LIN {X 0,Y 580.037,Z 775.595,A -85,B 0,C 180,E1 -1977.917,E2 -1977.917} C_VEL
LIN {X 0,Y 580.044,Z 776.896,A -85,B 0,C 180,E1 -1978.611,E2 -1978.611} C_VEL
LIN {X 0,Y 580.037,Z 777.71,A -85,B 0,C 180,E1 -1979.306,E2 -1979.306} C_VEL
LIN {X 0,Y 580.035,Z 777.996,A -85,B 0,C 180,E1 -1980,E2 -1980} C_VEL
LIN {X 0,Y 580.038,Z 777.754,A -85,B 0,C 180,E1 -1980.694,E2 -1980.694} C_VEL
LIN {X 0,Y 580.047,Z 777.018,A -85,B 0,C 180,E1 -1981.389,E2 -1981.389} C_VEL
LIN {X 0,Y 580.04,Z 775.802,A -85,B 0,C 180,E1 -1982.083,E2 -1982.083} C_VEL
LIN {X 0,Y 580.073,Z 772.961,A -85,B 0,C 180,E1 -1983.125,E2 -1983.125} C_VEL
LIN {X 0,Y 580.105,Z 768.85,A -85,B 0,C 180,E1 -1984.169,E2 -1984.169} C_VEL
LIN {X 0,Y 580.091,Z 763.255,A -85,B 0,C 180,E1 -1985.213,E2 -1985.213} C_VEL
LIN {X 0,Y 580.207,Z 757.174,A -85,B 0,C 180,E1 -1986.084,E2 -1986.084} C_VEL
LIN {X 0,Y 580.224,Z 749.516,A -85,B 0,C 180,E1 -1986.957,E2 -1986.957} C_VEL
LIN {X 0,Y 580.284,Z 740.89,A -85,B 0,C 180,E1 -1987.744,E2 -1987.744} C_VEL
LIN {X 0,Y 580.383,Z 731,A -85,B 0,C 180,E1 -1988.443,E2 -1988.443} C_VEL
LIN {X 0,Y 580.42,Z 721.403,A -85,B 0,C 180,E1 -1988.969,E2 -1988.969} C_VEL
LIN {X 0,Y 580.469,Z 711.987,A -85,B 0,C 180,E1 -1989.363,E2 -1989.363} C_VEL
LIN {X 0,Y 580.511,Z 701.019,A -85,B 0,C 180,E1 -1989.692,E2 -1989.692} C_VEL
LIN {X 0,Y 580.608,Z 688.344,A -85,B 0,C 180,E1 -1989.911,E2 -1989.911} C_VEL
LIN {X 0,Y 580.624,Z 626.629,A -85,B 0,C 180,E1 -1990.67,E2 -1990.67} C_VEL
LIN {X 0,Y 579.916,Z 622.77,A -85,B 0,C 180,E1 -1990.759,E2 -1990.759} C_VEL
LIN {X 0,Y 578.276,Z 619.333,A -85,B 0,C 180,E1 -1990.91,E2 -1990.91} C_VEL
LIN {X 0,Y 575.656,Z 615.329,A -85,B 0,C 180,E1 -1991.191,E2 -1991.191} C_VEL
LIN {X 0,Y 573.643,Z 611.693,A -85,B 0,C 180,E1 -1991.558,E2 -1991.558} C_VEL
LIN {X 0,Y 573.314,Z 609.974,A -85,B 0,C 180,E1 -1991.77,E2 -1991.77} C_VEL
LIN {X 0,Y 573.481,Z 588.417,A -85,B 0,C 180,E1 -1994.607,E2 -1994.607} C_VEL
LIN {X 0,Y 573.675,Z 565.715,A -85,B 0,C 180,E1 -1997.632,E2 -1997.632} C_VEL
LIN {X 0,Y 573.922,Z 545.049,A -85,B 0,C 180,E1 -2000.426,E2 -2000.426} C_VEL
LIN {X 0,Y 574.25,Z 522.477,A -85,B 0,C 180,E1 -2003.532,E2 -2003.532} C_VEL
LIN {X 0,Y 574.202,Z 517.675,A -85,B 0,C 180,E1 -2004.207,E2 -2004.207} C_VEL
LIN {X 0,Y 573.309,Z 513.19,A -85,B 0,C 180,E1 -2004.924,E2 -2004.924} C_VEL
LIN {X 0,Y 573.256,Z 513.08,A -85,B 0,C 180,E1 -2008.029,E2 -2008.029} C_VEL
LIN {X 0,Y 573.249,Z 513.077,A -85,B 0,C 180,E1 -2010.176,E2 -2010.176} C_VEL
LIN {X 0,Y 573.256,Z 513.073,A -85,B 0,C 180,E1 -2012.645,E2 -2012.645} C_VEL
LIN {X 0,Y 573.257,Z 513.076,A -85,B 0,C 180,E1 -2015.185,E2 -2015.185} C_VEL
LIN {X 0,Y 573.237,Z 513.08,A -85,B 0,C 180,E1 -2017.808,E2 -2017.808} C_VEL
LIN {X 0,Y 573.248,Z 513.07,A -85,B 0,C 180,E1 -2020.525,E2 -2020.525} C_VEL
LIN {X 0,Y 573.239,Z 513.077,A -85,B 0,C 180,E1 -2023.359,E2 -2023.359} C_VEL
LIN {X 0,Y 573.249,Z 513.073,A -85,B 0,C 180,E1 -2026.331,E2 -2026.331} C_VEL
LIN {X 0,Y 573.238,Z 513.074,A -85,B 0,C 180,E1 -2028.543,E2 -2028.543} C_VEL
LIN {X 0,Y 573.246,Z 513.081,A -85,B 0,C 180,E1 -2031.298,E2 -2031.298} C_VEL
LIN {X 0,Y 573.217,Z 513.077,A -85,B 0,C 180,E1 -2034.018,E2 -2034.018} C_VEL
LIN {X 0,Y 573.243,Z 513.075,A -85,B 0,C 180,E1 -2036.516,E2 -2036.516} C_VEL
LIN {X 0,Y 573.235,Z 513.084,A -85,B 0,C 180,E1 -2039.117,E2 -2039.117} C_VEL
LIN {X 0,Y 573.256,Z 513.073,A -85,B 0,C 180,E1 -2041.971,E2 -2041.971} C_VEL
LIN {X 0,Y 573.253,Z 513.079,A -85,B 0,C 180,E1 -2044.589,E2 -2044.589} C_VEL
LIN {X 0,Y 573.238,Z 513.075,A -85,B 0,C 180,E1 -2047.662,E2 -2047.662} C_VEL
LIN {X 0,Y 573.317,Z 513.261,A -85,B 0,C 180,E1 -2050.276,E2 -2050.276} C_VEL
LIN {X 0,Y 573.558,Z 518.552,A -85,B 0,C 180,E1 -2051.237,E2 -2051.237} C_VEL
LIN {X 0,Y 573.387,Z 536.372,A -85,B 0,C 180,E1 -2054.356,E2 -2054.356} C_VEL
LIN {X 0,Y 573.308,Z 547.196,A -85,B 0,C 180,E1 -2056.192,E2 -2056.192} C_VEL
LIN {X 0,Y 573.776,Z 550.138,A -85,B 0,C 180,E1 -2056.277,E2 -2056.277} C_VEL
LIN {X 0,Y 574.078,Z 556.843,A -85,B 0,C 180,E1 -2056.369,E2 -2056.369} C_VEL
LIN {X 0,Y 573.884,Z 653.915,A -85,B 0,C 180,E1 -2057.602,E2 -2057.602} C_VEL
LIN {X 0,Y 573.815,Z 667.201,A -85,B 0,C 180,E1 -2057.915,E2 -2057.915} C_VEL
LIN {X 0,Y 573.718,Z 679.36,A -85,B 0,C 180,E1 -2058.339,E2 -2058.339} C_VEL
LIN {X 0,Y 573.588,Z 690.955,A -85,B 0,C 180,E1 -2058.881,E2 -2058.881} C_VEL
LIN {X 0,Y 573.447,Z 702.546,A -85,B 0,C 180,E1 -2059.585,E2 -2059.585} C_VEL
LIN {X 0,Y 573.332,Z 713.058,A -85,B 0,C 180,E1 -2060.385,E2 -2060.385} C_VEL
LIN {X 0,Y 573.242,Z 721.659,A -85,B 0,C 180,E1 -2061.184,E2 -2061.184} C_VEL
LIN {X 0,Y 573.162,Z 729.583,A -85,B 0,C 180,E1 -2062.07,E2 -2062.07} C_VEL
LIN {X 0,Y 573.092,Z 737.519,A -85,B 0,C 180,E1 -2063.162,E2 -2063.162} C_VEL
LIN {X 0,Y 573.071,Z 744.447,A -85,B 0,C 180,E1 -2064.369,E2 -2064.369} C_VEL
LIN {X 0,Y 573.028,Z 749.189,A -85,B 0,C 180,E1 -2065.427,E2 -2065.427} C_VEL
LIN {X 0,Y 573.022,Z 752.822,A -85,B 0,C 180,E1 -2066.484,E2 -2066.484} C_VEL
LIN {X 0,Y 572.959,Z 754.699,A -85,B 0,C 180,E1 -2067.187,E2 -2067.187} C_VEL
LIN {X 0,Y 572.939,Z 756.128,A -85,B 0,C 180,E1 -2067.89,E2 -2067.89} C_VEL
LIN {X 0,Y 572.941,Z 757.755,A -85,B 0,C 180,E1 -2069.297,E2 -2069.297} C_VEL
LIN {X 0,Y 572.939,Z 757.996,A -85,B 0,C 180,E1 -2069.999,E2 -2069.999} C_VEL
LIN {X 0,Y 572.94,Z 757.815,A -85,B 0,C 180,E1 -2070.702,E2 -2070.702} C_VEL
LIN {X 0,Y 572.939,Z 756.273,A -85,B 0,C 180,E1 -2072.108,E2 -2072.108} C_VEL
LIN {X 0,Y 572.96,Z 754.912,A -85,B 0,C 180,E1 -2072.812,E2 -2072.812} C_VEL
LIN {X 0,Y 573.015,Z 752.034,A -85,B 0,C 180,E1 -2073.867,E2 -2073.867} C_VEL
LIN {X 0,Y 572.963,Z 748.134,A -85,B 0,C 180,E1 -2074.925,E2 -2074.925} C_VEL
LIN {X 0,Y 573.075,Z 743.102,A -85,B 0,C 180,E1 -2075.983,E2 -2075.983} C_VEL
LIN {X 0,Y 573.082,Z 736.781,A -85,B 0,C 180,E1 -2077.044,E2 -2077.044} C_VEL
LIN {X 0,Y 573.177,Z 728.86,A -85,B 0,C 180,E1 -2078.105,E2 -2078.105} C_VEL
LIN {X 0,Y 573.286,Z 719.011,A -85,B 0,C 180,E1 -2079.17,E2 -2079.17} C_VEL
LIN {X 0,Y 573.424,Z 708.694,A -85,B 0,C 180,E1 -2080.058,E2 -2080.058} C_VEL
LIN {X 0,Y 573.556,Z 697.058,A -85,B 0,C 180,E1 -2080.858,E2 -2080.858} C_VEL
LIN {X 0,Y 573.657,Z 686.212,A -85,B 0,C 180,E1 -2081.449,E2 -2081.449} C_VEL
LIN {X 0,Y 573.754,Z 673.632,A -85,B 0,C 180,E1 -2081.969,E2 -2081.969} C_VEL
LIN {X 0,Y 573.845,Z 660.474,A -85,B 0,C 180,E1 -2082.353,E2 -2082.353} C_VEL
LIN {X 0,Y 573.912,Z 648.141,A -85,B 0,C 180,E1 -2082.576,E2 -2082.576} C_VEL
LIN {X 0,Y 573.917,Z 551.106,A -85,B 0,C 180,E1 -2083.798,E2 -2083.798} C_VEL
LIN {X 0,Y 573.364,Z 547.542,A -85,B 0,C 180,E1 -2083.873,E2 -2083.873} C_VEL
LIN {X 0,Y 573.298,Z 546.336,A -85,B 0,C 180,E1 -2084.011,E2 -2084.011} C_VEL
LIN {X 0,Y 573.451,Z 530.701,A -85,B 0,C 180,E1 -2086.721,E2 -2086.721} C_VEL
LIN {X 0,Y 573.578,Z 515.71,A -85,B 0,C 180,E1 -2089.356,E2 -2089.356} C_VEL
LIN {X 0,Y 573.272,Z 513.184,A -85,B 0,C 180,E1 -2089.841,E2 -2089.841} C_VEL
LIN {X 0,Y 573.238,Z 513.076,A -85,B 0,C 180,E1 -2092.337,E2 -2092.337} C_VEL
LIN {X 0,Y 573.256,Z 513.081,A -85,B 0,C 180,E1 -2095.409,E2 -2095.409} C_VEL
LIN {X 0,Y 573.253,Z 513.074,A -85,B 0,C 180,E1 -2098.028,E2 -2098.028} C_VEL
LIN {X 0,Y 573.239,Z 513.076,A -85,B 0,C 180,E1 -2100.883,E2 -2100.883} C_VEL
LIN {X 0,Y 573.261,Z 513.08,A -85,B 0,C 180,E1 -2103.523,E2 -2103.523} C_VEL
LIN {X 0,Y 573.259,Z 513.072,A -85,B 0,C 180,E1 -2106.047,E2 -2106.047} C_VEL
LIN {X 0,Y 573.247,Z 513.074,A -85,B 0,C 180,E1 -2108.7,E2 -2108.7} C_VEL
LIN {X 0,Y 573.252,Z 513.08,A -85,B 0,C 180,E1 -2111.595,E2 -2111.595} C_VEL
LIN {X 0,Y 573.236,Z 513.073,A -85,B 0,C 180,E1 -2114.332,E2 -2114.332} C_VEL
LIN {X 0,Y 573.236,Z 513.083,A -85,B 0,C 180,E1 -2117.358,E2 -2117.358} C_VEL
LIN {X 0,Y 573.246,Z 513.071,A -85,B 0,C 180,E1 -2120.393,E2 -2120.393} C_VEL
LIN {X 0,Y 573.251,Z 513.075,A -85,B 0,C 180,E1 -2123.077,E2 -2123.077} C_VEL
LIN {X 0,Y 573.27,Z 513.077,A -85,B 0,C 180,E1 -2125.671,E2 -2125.671} C_VEL
LIN {X 0,Y 573.245,Z 513.074,A -85,B 0,C 180,E1 -2128.185,E2 -2128.185} C_VEL
LIN {X 0,Y 573.265,Z 513.071,A -85,B 0,C 180,E1 -2130.634,E2 -2130.634} C_VEL
LIN {X 0,Y 573.265,Z 513.08,A -85,B 0,C 180,E1 -2133.5,E2 -2133.5} C_VEL
LIN {X 0,Y 573.227,Z 513.076,A -85,B 0,C 180,E1 -2136.134,E2 -2136.134} C_VEL
LIN {X 0,Y 573.256,Z 513.076,A -85,B 0,C 180,E1 -2139.174,E2 -2139.174} C_VEL
LIN {X 0,Y 573.233,Z 513.083,A -85,B 0,C 180,E1 -2141.411,E2 -2141.411} C_VEL
LIN {X 0,Y 573.253,Z 513.08,A -85,B 0,C 180,E1 -2143.622,E2 -2143.622} C_VEL
LIN {X 0,Y 573.229,Z 513.075,A -85,B 0,C 180,E1 -2146.529,E2 -2146.529} C_VEL
LIN {X 0,Y 573.255,Z 513.072,A -85,B 0,C 180,E1 -2148.745,E2 -2148.745} C_VEL
LIN {X 0,Y 573.301,Z 513.075,A -85,B 0,C 180,E1 -2151.541,E2 -2151.541} C_VEL
LIN {X 0,Y 573.285,Z 513.068,A -85,B 0,C 180,E1 -2154.372,E2 -2154.372} C_VEL
LIN {X 0,Y 573.303,Z 513.07,A -85,B 0,C 180,E1 -2157.892,E2 -2157.892} C_VEL
LIN {X 0,Y 573.33,Z 513.063,A -85,B 0,C 180,E1 -2160.702,E2 -2160.702} C_VEL
LIN {X 0,Y 573.234,Z 513.083,A -85,B 0,C 180,E1 -2163.514,E2 -2163.514} C_VEL
LIN {X 0,Y 573.284,Z 513.078,A -85,B 0,C 180,E1 -2165.628,E2 -2165.628} C_VEL
LIN {X 0,Y 573.285,Z 513.068,A -85,B 0,C 180,E1 -2168.459,E2 -2168.459} C_VEL
LIN {X 0,Y 573.264,Z 513.075,A -85,B 0,C 180,E1 -2171.312,E2 -2171.312} C_VEL
LIN {X 0,Y 573.266,Z 513.072,A -85,B 0,C 180,E1 -2174.193,E2 -2174.193} C_VEL
LIN {X 0,Y 573.252,Z 513.074,A -85,B 0,C 180,E1 -2177.112,E2 -2177.112} C_VEL
LIN {X 0,Y 573.249,Z 513.075,A -85,B 0,C 180,E1 -2180.077,E2 -2180.077} C_VEL
LIN {X 0,Y 573.231,Z 513.075,A -85,B 0,C 180,E1 -2182.338,E2 -2182.338} C_VEL
LIN {X 0,Y 573.251,Z 513.079,A -85,B 0,C 180,E1 -2185.41,E2 -2185.41} C_VEL
LIN {X 0,Y 573.258,Z 513.076,A -85,B 0,C 180,E1 -2188.032,E2 -2188.032} C_VEL
LIN {X 0,Y 573.232,Z 513.075,A -85,B 0,C 180,E1 -2190.885,E2 -2190.885} C_VEL
LIN {X 0,Y 573.283,Z 513.077,A -85,B 0,C 180,E1 -2193.529,E2 -2193.529} C_VEL
LIN {X 0,Y 573.256,Z 513.073,A -85,B 0,C 180,E1 -2196.049,E2 -2196.049} C_VEL
LIN {X 0,Y 573.244,Z 513.073,A -85,B 0,C 180,E1 -2198.702,E2 -2198.702} C_VEL
LIN {X 0,Y 573.249,Z 513.082,A -85,B 0,C 180,E1 -2201.596,E2 -2201.596} C_VEL
LIN {X 0,Y 573.231,Z 513.076,A -85,B 0,C 180,E1 -2204.334,E2 -2204.334} C_VEL
LIN {X 0,Y 573.248,Z 513.077,A -85,B 0,C 180,E1 -2207.358,E2 -2207.358} C_VEL
LIN {X 0,Y 573.245,Z 513.073,A -85,B 0,C 180,E1 -2210.394,E2 -2210.394} C_VEL
LIN {X 0,Y 573.254,Z 513.071,A -85,B 0,C 180,E1 -2213.079,E2 -2213.079} C_VEL
LIN {X 0,Y 573.266,Z 513.08,A -85,B 0,C 180,E1 -2215.672,E2 -2215.672} C_VEL
LIN {X 0,Y 573.248,Z 513.065,A -85,B 0,C 180,E1 -2218.186,E2 -2218.186} C_VEL
LIN {X 0,Y 573.263,Z 513.071,A -85,B 0,C 180,E1 -2220.635,E2 -2220.635} C_VEL
LIN {X 0,Y 573.251,Z 513.073,A -85,B 0,C 180,E1 -2223.025,E2 -2223.025} C_VEL
LIN {X 0,Y 573.275,Z 513.075,A -85,B 0,C 180,E1 -2225.367,E2 -2225.367} C_VEL
LIN {X 0,Y 573.287,Z 513.31,A -85,B 0,C 180,E1 -2226.936,E2 -2226.936} C_VEL
LIN {X 0,Y 574.008,Z 518.026,A -85,B 0,C 180,E1 -2227.695,E2 -2227.695} C_VEL
LIN {X 0,Y 573.748,Z 538.175,A -85,B 0,C 180,E1 -2230.688,E2 -2230.688} C_VEL
LIN {X 0,Y 573.546,Z 557.107,A -85,B 0,C 180,E1 -2233.454,E2 -2233.454} C_VEL
LIN {X 0,Y 573.395,Z 576.024,A -85,B 0,C 180,E1 -2236.15,E2 -2236.15} C_VEL
LIN {X 0,Y 574.056,Z 581.566,A -85,B 0,C 180,E1 -2236.257,E2 -2236.257} C_VEL
LIN {X 0,Y 573.882,Z 683.982,A -85,B 0,C 180,E1 -2237.558,E2 -2237.558} C_VEL
LIN {X 0,Y 573.811,Z 697.238,A -85,B 0,C 180,E1 -2237.871,E2 -2237.871} C_VEL
LIN {X 0,Y 573.718,Z 709.387,A -85,B 0,C 180,E1 -2238.295,E2 -2238.295} C_VEL
LIN {X 0,Y 573.576,Z 721.729,A -85,B 0,C 180,E1 -2238.879,E2 -2238.879} C_VEL
LIN {X 0,Y 573.438,Z 733.213,A -85,B 0,C 180,E1 -2239.586,E2 -2239.586} C_VEL
LIN {X 0,Y 573.327,Z 743.607,A -85,B 0,C 180,E1 -2240.386,E2 -2240.386} C_VEL
LIN {X 0,Y 573.24,Z 752.119,A -85,B 0,C 180,E1 -2241.185,E2 -2241.185} C_VEL
LIN {X 0,Y 573.16,Z 759.966,A -85,B 0,C 180,E1 -2242.072,E2 -2242.072} C_VEL
LIN {X 0,Y 573.072,Z 767.958,A -85,B 0,C 180,E1 -2243.186,E2 -2243.186} C_VEL
LIN {X 0,Y 573.07,Z 774.683,A -85,B 0,C 180,E1 -2244.37,E2 -2244.37} C_VEL
LIN {X 0,Y 573.028,Z 779.374,A -85,B 0,C 180,E1 -2245.428,E2 -2245.428} C_VEL
LIN {X 0,Y 573.022,Z 782.96,A -85,B 0,C 180,E1 -2246.485,E2 -2246.485} C_VEL
LIN {X 0,Y 572.959,Z 784.811,A -85,B 0,C 180,E1 -2247.188,E2 -2247.188} C_VEL
LIN {X 0,Y 572.937,Z 786.201,A -85,B 0,C 180,E1 -2247.892,E2 -2247.892} C_VEL
LIN {X 0,Y 572.94,Z 787.785,A -85,B 0,C 180,E1 -2249.298,E2 -2249.298} C_VEL
LIN {X 0,Y 572.938,Z 788,A -85,B 0,C 180,E1 -2250.001,E2 -2250.001} C_VEL
LIN {X 0,Y 572.946,Z 787.185,A -85,B 0,C 180,E1 -2251.406,E2 -2251.406} C_VEL
LIN {X 0,Y 572.937,Z 786.198,A -85,B 0,C 180,E1 -2252.11,E2 -2252.11} C_VEL
LIN {X 0,Y 572.959,Z 784.807,A -85,B 0,C 180,E1 -2252.813,E2 -2252.813} C_VEL
LIN {X 0,Y 573.014,Z 781.894,A -85,B 0,C 180,E1 -2253.869,E2 -2253.869} C_VEL
LIN {X 0,Y 572.963,Z 777.948,A -85,B 0,C 180,E1 -2254.926,E2 -2254.926} C_VEL
LIN {X 0,Y 573.064,Z 771.874,A -85,B 0,C 180,E1 -2256.161,E2 -2256.161} C_VEL
LIN {X 0,Y 573.12,Z 765.234,A -85,B 0,C 180,E1 -2257.221,E2 -2257.221} C_VEL
LIN {X 0,Y 573.201,Z 756.986,A -85,B 0,C 180,E1 -2258.284,E2 -2258.284} C_VEL
LIN {X 0,Y 573.287,Z 748.532,A -85,B 0,C 180,E1 -2259.171,E2 -2259.171} C_VEL
LIN {X 0,Y 573.409,Z 738.091,A -85,B 0,C 180,E1 -2260.059,E2 -2260.059} C_VEL
LIN {X 0,Y 573.55,Z 726.343,A -85,B 0,C 180,E1 -2260.858,E2 -2260.858} C_VEL
LIN {X 0,Y 573.654,Z 715.271,A -85,B 0,C 180,E1 -2261.448,E2 -2261.448} C_VEL
LIN {X 0,Y 573.767,Z 702.163,A -85,B 0,C 180,E1 -2261.974,E2 -2261.974} C_VEL
LIN {X 0,Y 573.836,Z 689.501,A -85,B 0,C 180,E1 -2262.332,E2 -2262.332} C_VEL
LIN {X 0,Y 573.932,Z 676.268,A -85,B 0,C 180,E1 -2262.554,E2 -2262.554} C_VEL
LIN {X 0,Y 573.931,Z 579.679,A -85,B 0,C 180,E1 -2263.77,E2 -2263.77} C_VEL
LIN {X 0,Y 573.406,Z 576.004,A -85,B 0,C 180,E1 -2263.851,E2 -2263.851} C_VEL
LIN {X 0,Y 573.548,Z 555.884,A -85,B 0,C 180,E1 -2266.724,E2 -2266.724} C_VEL
LIN {X 0,Y 573.741,Z 537.567,A -85,B 0,C 180,E1 -2269.402,E2 -2269.402} C_VEL
LIN {X 0,Y 574.002,Z 518.017,A -85,B 0,C 180,E1 -2272.307,E2 -2272.307} C_VEL
LIN {X 0,Y 573.242,Z 513.207,A -85,B 0,C 180,E1 -2273.1,E2 -2273.1} C_VEL
LIN {X 0,Y 573.253,Z 513.074,A -85,B 0,C 180,E1 -2275.411,E2 -2275.411} C_VEL
LIN {X 0,Y 573.255,Z 513.08,A -85,B 0,C 180,E1 -2278.029,E2 -2278.029} C_VEL
LIN {X 0,Y 573.233,Z 513.077,A -85,B 0,C 180,E1 -2280.882,E2 -2280.882} C_VEL
LIN {X 0,Y 573.267,Z 513.072,A -85,B 0,C 180,E1 -2283.524,E2 -2283.524} C_VEL
LIN {X 0,Y 573.218,Z 513.084,A -85,B 0,C 180,E1 -2286.052,E2 -2286.052} C_VEL
LIN {X 0,Y 573.246,Z 513.077,A -85,B 0,C 180,E1 -2288.702,E2 -2288.702} C_VEL
LIN {X 0,Y 573.24,Z 513.076,A -85,B 0,C 180,E1 -2291.594,E2 -2291.594} C_VEL
LIN {X 0,Y 573.241,Z 513.083,A -85,B 0,C 180,E1 -2294.333,E2 -2294.333} C_VEL
LIN {X 0,Y 573.243,Z 513.074,A -85,B 0,C 180,E1 -2297.359,E2 -2297.359} C_VEL
LIN {X 0,Y 573.245,Z 513.081,A -85,B 0,C 180,E1 -2300.393,E2 -2300.393} C_VEL
LIN {X 0,Y 573.256,Z 513.073,A -85,B 0,C 180,E1 -2303.078,E2 -2303.078} C_VEL
LIN {X 0,Y 573.274,Z 513.073,A -85,B 0,C 180,E1 -2305.672,E2 -2305.672} C_VEL
LIN {X 0,Y 573.244,Z 513.084,A -85,B 0,C 180,E1 -2308.185,E2 -2308.185} C_VEL
LIN {X 0,Y 573.269,Z 513.075,A -85,B 0,C 180,E1 -2310.634,E2 -2310.634} C_VEL
LIN {X 0,Y 573.254,Z 513.075,A -85,B 0,C 180,E1 -2313.024,E2 -2313.024} C_VEL
LIN {X 0,Y 573.302,Z 513.274,A -85,B 0,C 180,E1 -2315.196,E2 -2315.196} C_VEL
LIN {X 0,Y 574.275,Z 518.402,A -85,B 0,C 180,E1 -2315.989,E2 -2315.989} C_VEL
LIN {X 0,Y 573.998,Z 537.56,A -85,B 0,C 180,E1 -2318.639,E2 -2318.639} C_VEL
LIN {X 0,Y 573.775,Z 556.702,A -85,B 0,C 180,E1 -2321.245,E2 -2321.245} C_VEL
LIN {X 0,Y 573.562,Z 577.222,A -85,B 0,C 180,E1 -2323.996,E2 -2323.996} C_VEL
LIN {X 0,Y 573.398,Z 599.11,A -85,B 0,C 180,E1 -2326.894,E2 -2326.894} C_VEL
LIN {X 0,Y 573.289,Z 616.348,A -85,B 0,C 180,E1 -2329.132,E2 -2329.132} C_VEL
LIN {X 0,Y 573.66,Z 621.84,A -85,B 0,C 180,E1 -2329.229,E2 -2329.229} C_VEL
LIN {X 0,Y 573.584,Z 695.63,A -85,B 0,C 180,E1 -2330.167,E2 -2330.167} C_VEL
LIN {X 0,Y 573.535,Z 706.772,A -85,B 0,C 180,E1 -2330.433,E2 -2330.433} C_VEL
LIN {X 0,Y 573.437,Z 717.591,A -85,B 0,C 180,E1 -2330.832,E2 -2330.832} C_VEL
LIN {X 0,Y 573.354,Z 728.01,A -85,B 0,C 180,E1 -2331.364,E2 -2331.364} C_VEL
LIN {X 0,Y 573.251,Z 737.417,A -85,B 0,C 180,E1 -2331.984,E2 -2331.984} C_VEL
LIN {X 0,Y 573.201,Z 746.873,A -85,B 0,C 180,E1 -2332.78,E2 -2332.78} C_VEL
LIN {X 0,Y 573.13,Z 755.029,A -85,B 0,C 180,E1 -2333.664,E2 -2333.664} C_VEL
LIN {X 0,Y 573.051,Z 761.518,A -85,B 0,C 180,E1 -2334.546,E2 -2334.546} C_VEL
LIN {X 0,Y 573.048,Z 766.692,A -85,B 0,C 180,E1 -2335.428,E2 -2335.428} C_VEL
LIN {X 0,Y 573.025,Z 771.452,A -85,B 0,C 180,E1 -2336.484,E2 -2336.484} C_VEL
LIN {X 0,Y 572.964,Z 773.816,A -85,B 0,C 180,E1 -2337.188,E2 -2337.188} C_VEL
LIN {X 0,Y 572.937,Z 775.601,A -85,B 0,C 180,E1 -2337.891,E2 -2337.891} C_VEL
LIN {X 0,Y 572.943,Z 776.902,A -85,B 0,C 180,E1 -2338.594,E2 -2338.594} C_VEL
LIN {X 0,Y 572.937,Z 777.711,A -85,B 0,C 180,E1 -2339.297,E2 -2339.297} C_VEL
LIN {X 0,Y 572.936,Z 777.996,A -85,B 0,C 180,E1 -2340,E2 -2340} C_VEL
LIN {X 0,Y 572.939,Z 777.759,A -85,B 0,C 180,E1 -2340.703,E2 -2340.703} C_VEL
LIN {X 0,Y 572.947,Z 777.022,A -85,B 0,C 180,E1 -2341.406,E2 -2341.406} C_VEL
LIN {X 0,Y 572.939,Z 775.805,A -85,B 0,C 180,E1 -2342.109,E2 -2342.109} C_VEL
LIN {X 0,Y 572.993,Z 772.965,A -85,B 0,C 180,E1 -2343.164,E2 -2343.164} C_VEL
LIN {X 0,Y 573.032,Z 768.854,A -85,B 0,C 180,E1 -2344.22,E2 -2344.22} C_VEL
LIN {X 0,Y 573.016,Z 763.251,A -85,B 0,C 180,E1 -2345.278,E2 -2345.278} C_VEL
LIN {X 0,Y 573.142,Z 757.176,A -85,B 0,C 180,E1 -2346.159,E2 -2346.159} C_VEL
LIN {X 0,Y 573.165,Z 749.518,A -85,B 0,C 180,E1 -2347.043,E2 -2347.043} C_VEL
LIN {X 0,Y 573.245,Z 740.886,A -85,B 0,C 180,E1 -2347.839,E2 -2347.839} C_VEL
LIN {X 0,Y 573.354,Z 730.997,A -85,B 0,C 180,E1 -2348.547,E2 -2348.547} C_VEL
LIN {X 0,Y 573.409,Z 721.406,A -85,B 0,C 180,E1 -2349.079,E2 -2349.079} C_VEL
LIN {X 0,Y 573.474,Z 711.987,A -85,B 0,C 180,E1 -2349.479,E2 -2349.479} C_VEL
LIN {X 0,Y 573.538,Z 701.001,A -85,B 0,C 180,E1 -2349.811,E2 -2349.811} C_VEL
LIN {X 0,Y 573.627,Z 688.299,A -85,B 0,C 180,E1 -2350.033,E2 -2350.033} C_VEL
LIN {X 0,Y 573.516,Z 618.508,A -85,B 0,C 180,E1 -2350.905,E2 -2350.905} C_VEL
LIN {X 0,Y 573.258,Z 616.098,A -85,B 0,C 180,E1 -2350.978,E2 -2350.978} C_VEL
LIN {X 0,Y 573.314,Z 609.974,A -85,B 0,C 180,E1 -2351.77,E2 -2351.77} C_VEL
LIN {X 0,Y 572.663,Z 606.483,A -85,B 0,C 180,E1 -2352.242,E2 -2352.242} C_VEL
LIN {X 0,Y 567.05,Z 595.597,A -85,B 0,C 180,E1 -2353.815,E2 -2353.815} C_VEL
LIN {X 0,Y 566.454,Z 592.116,A -85,B 0,C 180,E1 -2354.295,E2 -2354.295} C_VEL
LIN {X 0,Y 566.696,Z 568.311,A -85,B 0,C 180,E1 -2357.502,E2 -2357.502} C_VEL
LIN {X 0,Y 567.009,Z 546.413,A -85,B 0,C 180,E1 -2360.497,E2 -2360.497} C_VEL
LIN {X 0,Y 567.364,Z 524.423,A -85,B 0,C 180,E1 -2363.559,E2 -2363.559} C_VEL
LIN {X 0,Y 567.238,Z 518.888,A -85,B 0,C 180,E1 -2364.328,E2 -2364.328} C_VEL
LIN {X 0,Y 566.25,Z 514.044,A -85,B 0,C 180,E1 -2365.062,E2 -2365.062} C_VEL
LIN {X 0,Y 566.215,Z 513.955,A -85,B 0,C 180,E1 -2368.143,E2 -2368.143} C_VEL
LIN {X 0,Y 566.193,Z 513.955,A -85,B 0,C 180,E1 -2371.076,E2 -2371.076} C_VEL
LIN {X 0,Y 566.216,Z 513.958,A -85,B 0,C 180,E1 -2373.734,E2 -2373.734} C_VEL
LIN {X 0,Y 566.21,Z 513.95,A -85,B 0,C 180,E1 -2376.569,E2 -2376.569} C_VEL
LIN {X 0,Y 566.224,Z 513.952,A -85,B 0,C 180,E1 -2379.686,E2 -2379.686} C_VEL
LIN {X 0,Y 566.204,Z 513.946,A -85,B 0,C 180,E1 -2382.917,E2 -2382.917} C_VEL
LIN {X 0,Y 566.202,Z 513.952,A -85,B 0,C 180,E1 -2386.049,E2 -2386.049} C_VEL
LIN {X 0,Y 566.209,Z 513.956,A -85,B 0,C 180,E1 -2389.214,E2 -2389.214} C_VEL
LIN {X 0,Y 566.19,Z 513.955,A -85,B 0,C 180,E1 -2391.637,E2 -2391.637} C_VEL
LIN {X 0,Y 566.167,Z 513.956,A -85,B 0,C 180,E1 -2394.308,E2 -2394.308} C_VEL
LIN {X 0,Y 566.208,Z 513.957,A -85,B 0,C 180,E1 -2396.897,E2 -2396.897} C_VEL
LIN {X 0,Y 566.186,Z 513.957,A -85,B 0,C 180,E1 -2399.407,E2 -2399.407} C_VEL
LIN {X 0,Y 566.217,Z 513.95,A -85,B 0,C 180,E1 -2401.857,E2 -2401.857} C_VEL
LIN {X 0,Y 566.214,Z 513.952,A -85,B 0,C 180,E1 -2404.251,E2 -2404.251} C_VEL
LIN {X 0,Y 566.174,Z 513.962,A -85,B 0,C 180,E1 -2406.719,E2 -2406.719} C_VEL
LIN {X 0,Y 566.222,Z 513.956,A -85,B 0,C 180,E1 -2409.663,E2 -2409.663} C_VEL
LIN {X 0,Y 566.288,Z 514.172,A -85,B 0,C 180,E1 -2410.186,E2 -2410.186} C_VEL
LIN {X 0,Y 566.542,Z 520.652,A -85,B 0,C 180,E1 -2411.371,E2 -2411.371} C_VEL
LIN {X 0,Y 566.352,Z 537.424,A -85,B 0,C 180,E1 -2414.341,E2 -2414.341} C_VEL
LIN {X 0,Y 566.278,Z 547.213,A -85,B 0,C 180,E1 -2416.017,E2 -2416.017} C_VEL
LIN {X 0,Y 566.867,Z 550.854,A -85,B 0,C 180,E1 -2416.115,E2 -2416.115} C_VEL
LIN {X 0,Y 567.18,Z 556.888,A -85,B 0,C 180,E1 -2416.2,E2 -2416.2} C_VEL
LIN {X 0,Y 566.964,Z 653.944,A -85,B 0,C 180,E1 -2417.448,E2 -2417.448} C_VEL
LIN {X 0,Y 566.877,Z 667.22,A -85,B 0,C 180,E1 -2417.764,E2 -2417.764} C_VEL
LIN {X 0,Y 566.75,Z 679.376,A -85,B 0,C 180,E1 -2418.193,E2 -2418.193} C_VEL
LIN {X 0,Y 566.606,Z 691.637,A -85,B 0,C 180,E1 -2418.78,E2 -2418.78} C_VEL
LIN {X 0,Y 566.438,Z 703.842,A -85,B 0,C 180,E1 -2419.545,E2 -2419.545} C_VEL
LIN {X 0,Y 566.299,Z 714.125,A -85,B 0,C 180,E1 -2420.355,E2 -2420.355} C_VEL
LIN {X 0,Y 566.183,Z 723.374,A -85,B 0,C 180,E1 -2421.253,E2 -2421.253} C_VEL
LIN {X 0,Y 566.082,Z 732.345,A -85,B 0,C 180,E1 -2422.33,E2 -2422.33} C_VEL
LIN {X 0,Y 566.01,Z 739.456,A -85,B 0,C 180,E1 -2423.386,E2 -2423.386} C_VEL
LIN {X 0,Y 566.004,Z 744.449,A -85,B 0,C 180,E1 -2424.299,E2 -2424.299} C_VEL
LIN {X 0,Y 565.933,Z 749.191,A -85,B 0,C 180,E1 -2425.369,E2 -2425.369} C_VEL
LIN {X 0,Y 565.927,Z 752.824,A -85,B 0,C 180,E1 -2426.439,E2 -2426.439} C_VEL
LIN {X 0,Y 565.878,Z 754.701,A -85,B 0,C 180,E1 -2427.152,E2 -2427.152} C_VEL
LIN {X 0,Y 565.84,Z 756.128,A -85,B 0,C 180,E1 -2427.864,E2 -2427.864} C_VEL
LIN {X 0,Y 565.841,Z 757.755,A -85,B 0,C 180,E1 -2429.288,E2 -2429.288} C_VEL
LIN {X 0,Y 565.839,Z 757.996,A -85,B 0,C 180,E1 -2429.999,E2 -2429.999} C_VEL
LIN {X 0,Y 565.841,Z 757.815,A -85,B 0,C 180,E1 -2430.711,E2 -2430.711} C_VEL
LIN {X 0,Y 565.84,Z 756.272,A -85,B 0,C 180,E1 -2432.135,E2 -2432.135} C_VEL
LIN {X 0,Y 565.878,Z 754.911,A -85,B 0,C 180,E1 -2432.847,E2 -2432.847} C_VEL
LIN {X 0,Y 565.927,Z 752.032,A -85,B 0,C 180,E1 -2433.916,E2 -2433.916} C_VEL
LIN {X 0,Y 565.878,Z 748.132,A -85,B 0,C 180,E1 -2434.987,E2 -2434.987} C_VEL
LIN {X 0,Y 565.99,Z 743.1,A -85,B 0,C 180,E1 -2436.058,E2 -2436.058} C_VEL
LIN {X 0,Y 566.03,Z 736.777,A -85,B 0,C 180,E1 -2437.132,E2 -2437.132} C_VEL
LIN {X 0,Y 566.132,Z 728.855,A -85,B 0,C 180,E1 -2438.207,E2 -2438.207} C_VEL
LIN {X 0,Y 566.249,Z 719.005,A -85,B 0,C 180,E1 -2439.285,E2 -2439.285} C_VEL
LIN {X 0,Y 566.424,Z 708.688,A -85,B 0,C 180,E1 -2440.183,E2 -2440.183} C_VEL
LIN {X 0,Y 566.562,Z 697.411,A -85,B 0,C 180,E1 -2440.971,E2 -2440.971} C_VEL
LIN {X 0,Y 566.687,Z 686.2,A -85,B 0,C 180,E1 -2441.591,E2 -2441.591} C_VEL
LIN {X 0,Y 566.816,Z 673.618,A -85,B 0,C 180,E1 -2442.118,E2 -2442.118} C_VEL
LIN {X 0,Y 566.935,Z 660.451,A -85,B 0,C 180,E1 -2442.506,E2 -2442.506} C_VEL
LIN {X 0,Y 566.998,Z 648.1,A -85,B 0,C 180,E1 -2442.732,E2 -2442.732} C_VEL
LIN {X 0,Y 567.094,Z 552.181,A -85,B 0,C 180,E1 -2443.953,E2 -2443.953} C_VEL
LIN {X 0,Y 566.306,Z 547.546,A -85,B 0,C 180,E1 -2444.05,E2 -2444.05} C_VEL
LIN {X 0,Y 566.272,Z 546.336,A -85,B 0,C 180,E1 -2444.188,E2 -2444.188} C_VEL
LIN {X 0,Y 566.442,Z 529.292,A -85,B 0,C 180,E1 -2447.183,E2 -2447.183} C_VEL
LIN {X 0,Y 566.526,Z 515.918,A -85,B 0,C 180,E1 -2449.568,E2 -2449.568} C_VEL
LIN {X 0,Y 566.236,Z 514.029,A -85,B 0,C 180,E1 -2449.957,E2 -2449.957} C_VEL
LIN {X 0,Y 566.18,Z 513.956,A -85,B 0,C 180,E1 -2452.631,E2 -2452.631} C_VEL
LIN {X 0,Y 566.218,Z 513.954,A -85,B 0,C 180,E1 -2455.029,E2 -2455.029} C_VEL
LIN {X 0,Y 566.212,Z 513.958,A -85,B 0,C 180,E1 -2457.338,E2 -2457.338} C_VEL
LIN {X 0,Y 566.202,Z 513.954,A -85,B 0,C 180,E1 -2459.768,E2 -2459.768} C_VEL
LIN {X 0,Y 566.206,Z 513.95,A -85,B 0,C 180,E1 -2462.43,E2 -2462.43} C_VEL
LIN {X 0,Y 566.21,Z 513.954,A -85,B 0,C 180,E1 -2464.993,E2 -2464.993} C_VEL
LIN {X 0,Y 566.195,Z 513.961,A -85,B 0,C 180,E1 -2467.46,E2 -2467.46} C_VEL
LIN {X 0,Y 566.225,Z 513.947,A -85,B 0,C 180,E1 -2470.196,E2 -2470.196} C_VEL
LIN {X 0,Y 566.203,Z 513.955,A -85,B 0,C 180,E1 -2473.053,E2 -2473.053} C_VEL
LIN {X 0,Y 566.194,Z 513.953,A -85,B 0,C 180,E1 -2476.048,E2 -2476.048} C_VEL
LIN {X 0,Y 566.208,Z 513.952,A -85,B 0,C 180,E1 -2478.863,E2 -2478.863} C_VEL
LIN {X 0,Y 566.186,Z 513.958,A -85,B 0,C 180,E1 -2481.637,E2 -2481.637} C_VEL
LIN {X 0,Y 566.208,Z 513.95,A -85,B 0,C 180,E1 -2484.311,E2 -2484.311} C_VEL
LIN {X 0,Y 566.224,Z 513.95,A -85,B 0,C 180,E1 -2486.898,E2 -2486.898} C_VEL
LIN {X 0,Y 566.189,Z 513.961,A -85,B 0,C 180,E1 -2489.408,E2 -2489.408} C_VEL
LIN {X 0,Y 566.222,Z 513.951,A -85,B 0,C 180,E1 -2491.858,E2 -2491.858} C_VEL
LIN {X 0,Y 566.221,Z 513.949,A -85,B 0,C 180,E1 -2494.251,E2 -2494.251} C_VEL
LIN {X 0,Y 566.186,Z 513.953,A -85,B 0,C 180,E1 -2496.713,E2 -2496.713} C_VEL
LIN {X 0,Y 566.214,Z 513.956,A -85,B 0,C 180,E1 -2499.663,E2 -2499.663} C_VEL
LIN {X 0,Y 566.198,Z 513.95,A -85,B 0,C 180,E1 -2502.668,E2 -2502.668} C_VEL
LIN {X 0,Y 566.227,Z 513.956,A -85,B 0,C 180,E1 -2505.627,E2 -2505.627} C_VEL
LIN {X 0,Y 566.227,Z 513.947,A -85,B 0,C 180,E1 -2508.675,E2 -2508.675} C_VEL
LIN {X 0,Y 566.241,Z 513.952,A -85,B 0,C 180,E1 -2511.434,E2 -2511.434} C_VEL
LIN {X 0,Y 566.253,Z 513.945,A -85,B 0,C 180,E1 -2514.302,E2 -2514.302} C_VEL
LIN {X 0,Y 566.274,Z 513.946,A -85,B 0,C 180,E1 -2517.866,E2 -2517.866} C_VEL
LIN {X 0,Y 566.3,Z 513.939,A -85,B 0,C 180,E1 -2520.711,E2 -2520.711} C_VEL
LIN {X 0,Y 566.272,Z 513.941,A -85,B 0,C 180,E1 -2522.846,E2 -2522.846} C_VEL
LIN {X 0,Y 566.252,Z 513.952,A -85,B 0,C 180,E1 -2525.698,E2 -2525.698} C_VEL
LIN {X 0,Y 566.228,Z 513.947,A -85,B 0,C 180,E1 -2528.566,E2 -2528.566} C_VEL
LIN {X 0,Y 566.234,Z 513.953,A -85,B 0,C 180,E1 -2531.454,E2 -2531.454} C_VEL
LIN {X 0,Y 566.227,Z 513.947,A -85,B 0,C 180,E1 -2534.507,E2 -2534.507} C_VEL
LIN {X 0,Y 566.197,Z 513.955,A -85,B 0,C 180,E1 -2537.332,E2 -2537.332} C_VEL
LIN {X 0,Y 566.212,Z 513.949,A -85,B 0,C 180,E1 -2540.337,E2 -2540.337} C_VEL
LIN {X 0,Y 566.183,Z 513.959,A -85,B 0,C 180,E1 -2543.404,E2 -2543.404} C_VEL
LIN {X 0,Y 566.22,Z 513.955,A -85,B 0,C 180,E1 -2545.749,E2 -2545.749} C_VEL
LIN {X 0,Y 566.2,Z 513.953,A -85,B 0,C 180,E1 -2548.204,E2 -2548.204} C_VEL
LIN {X 0,Y 566.193,Z 513.953,A -85,B 0,C 180,E1 -2551.079,E2 -2551.079} C_VEL
LIN {X 0,Y 566.217,Z 513.953,A -85,B 0,C 180,E1 -2553.956,E2 -2553.956} C_VEL
LIN {X 0,Y 566.211,Z 513.946,A -85,B 0,C 180,E1 -2556.569,E2 -2556.569} C_VEL
LIN {X 0,Y 566.208,Z 513.96,A -85,B 0,C 180,E1 -2559.686,E2 -2559.686} C_VEL
LIN {X 0,Y 566.209,Z 513.951,A -85,B 0,C 180,E1 -2562.088,E2 -2562.088} C_VEL
LIN {X 0,Y 566.169,Z 513.956,A -85,B 0,C 180,E1 -2565.037,E2 -2565.037} C_VEL
LIN {X 0,Y 566.214,Z 513.956,A -85,B 0,C 180,E1 -2567.914,E2 -2567.914} C_VEL
LIN {X 0,Y 566.219,Z 513.947,A -85,B 0,C 180,E1 -2570.728,E2 -2570.728} C_VEL
LIN {X 0,Y 566.204,Z 513.96,A -85,B 0,C 180,E1 -2573.786,E2 -2573.786} C_VEL
LIN {X 0,Y 566.228,Z 513.946,A -85,B 0,C 180,E1 -2576.899,E2 -2576.899} C_VEL
LIN {X 0,Y 566.187,Z 513.945,A -85,B 0,C 180,E1 -2579.409,E2 -2579.409} C_VEL
LIN {X 0,Y 566.228,Z 513.955,A -85,B 0,C 180,E1 -2581.859,E2 -2581.859} C_VEL
LIN {X 0,Y 566.213,Z 513.95,A -85,B 0,C 180,E1 -2584.252,E2 -2584.252} C_VEL
LIN {X 0,Y 566.212,Z 514.098,A -85,B 0,C 180,E1 -2586.741,E2 -2586.741} C_VEL
LIN {X 0,Y 567.096,Z 519.285,A -85,B 0,C 180,E1 -2587.6,E2 -2587.6} C_VEL
LIN {X 0,Y 566.788,Z 539.048,A -85,B 0,C 180,E1 -2590.571,E2 -2590.571} C_VEL
LIN {X 0,Y 566.562,Z 557.208,A -85,B 0,C 180,E1 -2593.259,E2 -2593.259} C_VEL
LIN {X 0,Y 566.406,Z 576.031,A -85,B 0,C 180,E1 -2595.976,E2 -2595.976} C_VEL
LIN {X 0,Y 567.174,Z 582.359,A -85,B 0,C 180,E1 -2596.097,E2 -2596.097} C_VEL
LIN {X 0,Y 566.972,Z 683.981,A -85,B 0,C 180,E1 -2597.404,E2 -2597.404} C_VEL
LIN {X 0,Y 566.866,Z 697.237,A -85,B 0,C 180,E1 -2597.72,E2 -2597.72} C_VEL
LIN {X 0,Y 566.762,Z 709.388,A -85,B 0,C 180,E1 -2598.149,E2 -2598.149} C_VEL
LIN {X 0,Y 566.626,Z 721.167,A -85,B 0,C 180,E1 -2598.709,E2 -2598.709} C_VEL
LIN {X 0,Y 566.459,Z 733.211,A -85,B 0,C 180,E1 -2599.456,E2 -2599.456} C_VEL
LIN {X 0,Y 566.319,Z 743.608,A -85,B 0,C 180,E1 -2600.266,E2 -2600.266} C_VEL
LIN {X 0,Y 566.207,Z 752.12,A -85,B 0,C 180,E1 -2601.075,E2 -2601.075} C_VEL
LIN {X 0,Y 566.112,Z 759.966,A -85,B 0,C 180,E1 -2601.972,E2 -2601.972} C_VEL
LIN {X 0,Y 566.003,Z 767.626,A -85,B 0,C 180,E1 -2603.047,E2 -2603.047} C_VEL
LIN {X 0,Y 566.003,Z 774.683,A -85,B 0,C 180,E1 -2604.3,E2 -2604.3} C_VEL
LIN {X 0,Y 565.933,Z 779.374,A -85,B 0,C 180,E1 -2605.371,E2 -2605.371} C_VEL
LIN {X 0,Y 565.927,Z 782.961,A -85,B 0,C 180,E1 -2606.441,E2 -2606.441} C_VEL
LIN {X 0,Y 565.878,Z 784.811,A -85,B 0,C 180,E1 -2607.153,E2 -2607.153} C_VEL
LIN {X 0,Y 565.846,Z 787.187,A -85,B 0,C 180,E1 -2608.577,E2 -2608.577} C_VEL
LIN {X 0,Y 565.839,Z 788,A -85,B 0,C 180,E1 -2610.001,E2 -2610.001} C_VEL
LIN {X 0,Y 565.846,Z 787.185,A -85,B 0,C 180,E1 -2611.424,E2 -2611.424} C_VEL
LIN {X 0,Y 565.878,Z 784.807,A -85,B 0,C 180,E1 -2612.848,E2 -2612.848} C_VEL
LIN {X 0,Y 565.926,Z 781.893,A -85,B 0,C 180,E1 -2613.917,E2 -2613.917} C_VEL
LIN {X 0,Y 565.878,Z 777.948,A -85,B 0,C 180,E1 -2614.988,E2 -2614.988} C_VEL
LIN {X 0,Y 566.002,Z 772.864,A -85,B 0,C 180,E1 -2616.059,E2 -2616.059} C_VEL
LIN {X 0,Y 566.041,Z 766.464,A -85,B 0,C 180,E1 -2617.133,E2 -2617.133} C_VEL
LIN {X 0,Y 566.134,Z 758.474,A -85,B 0,C 180,E1 -2618.208,E2 -2618.208} C_VEL
LIN {X 0,Y 566.229,Z 750.33,A -85,B 0,C 180,E1 -2619.106,E2 -2619.106} C_VEL
LIN {X 0,Y 566.339,Z 740.395,A -85,B 0,C 180,E1 -2620.005,E2 -2620.005} C_VEL
LIN {X 0,Y 566.526,Z 729.279,A -85,B 0,C 180,E1 -2620.808,E2 -2620.808} C_VEL
LIN {X 0,Y 566.614,Z 718.166,A -85,B 0,C 180,E1 -2621.447,E2 -2621.447} C_VEL
LIN {X 0,Y 566.75,Z 705.976,A -85,B 0,C 180,E1 -2621.988,E2 -2621.988} C_VEL
LIN {X 0,Y 566.916,Z 693.161,A -85,B 0,C 180,E1 -2622.394,E2 -2622.394} C_VEL
LIN {X 0,Y 566.992,Z 679.566,A -85,B 0,C 180,E1 -2622.665,E2 -2622.665} C_VEL
LIN {X 0,Y 567.033,Z 580.381,A -85,B 0,C 180,E1 -2623.932,E2 -2623.932} C_VEL
LIN {X 0,Y 566.399,Z 576.011,A -85,B 0,C 180,E1 -2624.026,E2 -2624.026} C_VEL
LIN {X 0,Y 566.573,Z 556.083,A -85,B 0,C 180,E1 -2626.906,E2 -2626.906} C_VEL
LIN {X 0,Y 566.83,Z 536.907,A -85,B 0,C 180,E1 -2629.747,E2 -2629.747} C_VEL
LIN {X 0,Y 567.078,Z 519.277,A -85,B 0,C 180,E1 -2632.402,E2 -2632.402} C_VEL
LIN {X 0,Y 566.189,Z 514.054,A -85,B 0,C 180,E1 -2633.285,E2 -2633.285} C_VEL
LIN {X 0,Y 566.214,Z 513.952,A -85,B 0,C 180,E1 -2635.749,E2 -2635.749} C_VEL
LIN {X 0,Y 566.207,Z 513.956,A -85,B 0,C 180,E1 -2638.202,E2 -2638.202} C_VEL
LIN {X 0,Y 566.195,Z 513.953,A -85,B 0,C 180,E1 -2641.077,E2 -2641.077} C_VEL
LIN {X 0,Y 566.216,Z 513.952,A -85,B 0,C 180,E1 -2643.734,E2 -2643.734} C_VEL
LIN {X 0,Y 566.203,Z 513.956,A -85,B 0,C 180,E1 -2646.57,E2 -2646.57} C_VEL
LIN {X 0,Y 566.219,Z 513.951,A -85,B 0,C 180,E1 -2649.686,E2 -2649.686} C_VEL
LIN {X 0,Y 566.209,Z 513.952,A -85,B 0,C 180,E1 -2652.918,E2 -2652.918} C_VEL
LIN {X 0,Y 566.197,Z 513.959,A -85,B 0,C 180,E1 -2656.049,E2 -2656.049} C_VEL
LIN {X 0,Y 566.207,Z 513.95,A -85,B 0,C 180,E1 -2659.215,E2 -2659.215} C_VEL
LIN {X 0,Y 566.191,Z 513.955,A -85,B 0,C 180,E1 -2661.637,E2 -2661.637} C_VEL
LIN {X 0,Y 566.197,Z 513.961,A -85,B 0,C 180,E1 -2664.31,E2 -2664.31} C_VEL
LIN {X 0,Y 566.223,Z 513.95,A -85,B 0,C 180,E1 -2666.898,E2 -2666.898} C_VEL
LIN {X 0,Y 566.183,Z 513.955,A -85,B 0,C 180,E1 -2669.407,E2 -2669.407} C_VEL
LIN {X 0,Y 566.233,Z 513.953,A -85,B 0,C 180,E1 -2671.858,E2 -2671.858} C_VEL
LIN {X 0,Y 566.219,Z 513.959,A -85,B 0,C 180,E1 -2674.251,E2 -2674.251} C_VEL
LIN {X 0,Y 566.267,Z 514.174,A -85,B 0,C 180,E1 -2675.114,E2 -2675.114} C_VEL
LIN {X 0,Y 567.386,Z 520.906,A -85,B 0,C 180,E1 -2676.047,E2 -2676.047} C_VEL
LIN {X 0,Y 567.053,Z 540.605,A -85,B 0,C 180,E1 -2678.788,E2 -2678.788} C_VEL
LIN {X 0,Y 566.79,Z 560.811,A -85,B 0,C 180,E1 -2681.567,E2 -2681.567} C_VEL
LIN {X 0,Y 566.522,Z 581.33,A -85,B 0,C 180,E1 -2684.346,E2 -2684.346} C_VEL
LIN {X 0,Y 566.358,Z 601.85,A -85,B 0,C 180,E1 -2687.093,E2 -2687.093} C_VEL
LIN {X 0,Y 566.225,Z 616.325,A -85,B 0,C 180,E1 -2688.992,E2 -2688.992} C_VEL
LIN {X 0,Y 566.708,Z 622.505,A -85,B 0,C 180,E1 -2689.104,E2 -2689.104} C_VEL
LIN {X 0,Y 566.595,Z 695.7,A -85,B 0,C 180,E1 -2690.045,E2 -2690.045} C_VEL
LIN {X 0,Y 566.528,Z 706.784,A -85,B 0,C 180,E1 -2690.314,E2 -2690.314} C_VEL
LIN {X 0,Y 566.438,Z 717.601,A -85,B 0,C 180,E1 -2690.718,E2 -2690.718} C_VEL
LIN {X 0,Y 566.338,Z 728.027,A -85,B 0,C 180,E1 -2691.256,E2 -2691.256} C_VEL
LIN {X 0,Y 566.206,Z 737.435,A -85,B 0,C 180,E1 -2691.883,E2 -2691.883} C_VEL
LIN {X 0,Y 566.141,Z 746.875,A -85,B 0,C 180,E1 -2692.69,E2 -2692.69} C_VEL
LIN {X 0,Y 566.072,Z 755.039,A -85,B 0,C 180,E1 -2693.584,E2 -2693.584} C_VEL
LIN {X 0,Y 565.986,Z 761.529,A -85,B 0,C 180,E1 -2694.478,E2 -2694.478} C_VEL
LIN {X 0,Y 565.973,Z 766.701,A -85,B 0,C 180,E1 -2695.37,E2 -2695.37} C_VEL
LIN {X 0,Y 565.932,Z 771.454,A -85,B 0,C 180,E1 -2696.44,E2 -2696.44} C_VEL
LIN {X 0,Y 565.883,Z 773.821,A -85,B 0,C 180,E1 -2697.153,E2 -2697.153} C_VEL
LIN {X 0,Y 565.839,Z 775.607,A -85,B 0,C 180,E1 -2697.865,E2 -2697.865} C_VEL
LIN {X 0,Y 565.843,Z 776.908,A -85,B 0,C 180,E1 -2698.577,E2 -2698.577} C_VEL
LIN {X 0,Y 565.838,Z 777.712,A -85,B 0,C 180,E1 -2699.288,E2 -2699.288} C_VEL
LIN {X 0,Y 565.837,Z 777.996,A -85,B 0,C 180,E1 -2700,E2 -2700} C_VEL
LIN {X 0,Y 565.839,Z 777.764,A -85,B 0,C 180,E1 -2700.712,E2 -2700.712} C_VEL
LIN {X 0,Y 565.846,Z 777.027,A -85,B 0,C 180,E1 -2701.423,E2 -2701.423} C_VEL
LIN {X 0,Y 565.841,Z 775.805,A -85,B 0,C 180,E1 -2702.135,E2 -2702.135} C_VEL
LIN {X 0,Y 565.914,Z 772.969,A -85,B 0,C 180,E1 -2703.204,E2 -2703.204} C_VEL
LIN {X 0,Y 565.962,Z 768.857,A -85,B 0,C 180,E1 -2704.273,E2 -2704.273} C_VEL
LIN {X 0,Y 565.946,Z 763.248,A -85,B 0,C 180,E1 -2705.344,E2 -2705.344} C_VEL
LIN {X 0,Y 566.078,Z 757.178,A -85,B 0,C 180,E1 -2706.237,E2 -2706.237} C_VEL
LIN {X 0,Y 566.117,Z 749.521,A -85,B 0,C 180,E1 -2707.131,E2 -2707.131} C_VEL
LIN {X 0,Y 566.182,Z 740.881,A -85,B 0,C 180,E1 -2707.938,E2 -2707.938} C_VEL
LIN {X 0,Y 566.334,Z 730.995,A -85,B 0,C 180,E1 -2708.654,E2 -2708.654} C_VEL
LIN {X 0,Y 566.409,Z 721.409,A -85,B 0,C 180,E1 -2709.193,E2 -2709.193} C_VEL
LIN {X 0,Y 566.509,Z 710.784,A -85,B 0,C 180,E1 -2709.641,E2 -2709.641} C_VEL
LIN {X 0,Y 566.559,Z 699.155,A -85,B 0,C 180,E1 -2709.979,E2 -2709.979} C_VEL
LIN {X 0,Y 566.61,Z 684.675,A -85,B 0,C 180,E1 -2710.203,E2 -2710.203} C_VEL
LIN {X 0,Y 566.616,Z 619.494,A -85,B 0,C 180,E1 -2711.026,E2 -2711.026} C_VEL
LIN {X 0,Y 566.232,Z 616.324,A -85,B 0,C 180,E1 -2711.098,E2 -2711.098} C_VEL
LIN {X 0,Y 566.433,Z 594.314,A -85,B 0,C 180,E1 -2714.002,E2 -2714.002} C_VEL
LIN {X 0,Y 566.454,Z 592.116,A -85,B 0,C 180,E1 -2714.295,E2 -2714.295} C_VEL
LIN {X 0,Y 565.843,Z 588.656,A -85,B 0,C 180,E1 -2714.776,E2 -2714.776} C_VEL
LIN {X 0,Y 560.223,Z 577.978,A -85,B 0,C 180,E1 -2716.383,E2 -2716.383} C_VEL
LIN {X 0,Y 559.65,Z 574.533,A -85,B 0,C 180,E1 -2716.873,E2 -2716.873} C_VEL
LIN {X 0,Y 560.036,Z 551.883,A -85,B 0,C 180,E1 -2719.997,E2 -2719.997} C_VEL
LIN {X 0,Y 560.327,Z 531.166,A -85,B 0,C 180,E1 -2722.881,E2 -2722.881} C_VEL
LIN {X 0,Y 560.401,Z 521.243,A -85,B 0,C 180,E1 -2724.25,E2 -2724.25} C_VEL
LIN {X 0,Y 559.218,Z 514.913,A -85,B 0,C 180,E1 -2725.195,E2 -2725.195} C_VEL
LIN {X 0,Y 559.185,Z 514.835,A -85,B 0,C 180,E1 -2727.712,E2 -2727.712} C_VEL
LIN {X 0,Y 559.156,Z 514.833,A -85,B 0,C 180,E1 -2730.183,E2 -2730.183} C_VEL
LIN {X 0,Y 559.16,Z 514.829,A -85,B 0,C 180,E1 -2732.715,E2 -2732.715} C_VEL
LIN {X 0,Y 559.148,Z 514.835,A -85,B 0,C 180,E1 -2735.323,E2 -2735.323} C_VEL
LIN {X 0,Y 559.136,Z 514.834,A -85,B 0,C 180,E1 -2738.018,E2 -2738.018} C_VEL
LIN {X 0,Y 559.159,Z 514.826,A -85,B 0,C 180,E1 -2740.812,E2 -2740.812} C_VEL
LIN {X 0,Y 559.142,Z 514.833,A -85,B 0,C 180,E1 -2743.734,E2 -2743.734} C_VEL
LIN {X 0,Y 559.151,Z 514.832,A -85,B 0,C 180,E1 -2746.803,E2 -2746.803} C_VEL
LIN {X 0,Y 559.161,Z 514.834,A -85,B 0,C 180,E1 -2749.188,E2 -2749.188} C_VEL
LIN {X 0,Y 559.137,Z 514.831,A -85,B 0,C 180,E1 -2751.982,E2 -2751.982} C_VEL
LIN {X 0,Y 559.136,Z 514.836,A -85,B 0,C 180,E1 -2754.787,E2 -2754.787} C_VEL
LIN {X 0,Y 559.158,Z 514.833,A -85,B 0,C 180,E1 -2757.365,E2 -2757.365} C_VEL
LIN {X 0,Y 559.153,Z 514.83,A -85,B 0,C 180,E1 -2760.142,E2 -2760.142} C_VEL
LIN {X 0,Y 559.174,Z 514.834,A -85,B 0,C 180,E1 -2763.097,E2 -2763.097} C_VEL
LIN {X 0,Y 559.16,Z 514.828,A -85,B 0,C 180,E1 -2765.495,E2 -2765.495} C_VEL
LIN {X 0,Y 559.177,Z 514.833,A -85,B 0,C 180,E1 -2768.624,E2 -2768.624} C_VEL
LIN {X 0,Y 559.235,Z 514.989,A -85,B 0,C 180,E1 -2770.069,E2 -2770.069} C_VEL
LIN {X 0,Y 559.557,Z 520.655,A -85,B 0,C 180,E1 -2771.13,E2 -2771.13} C_VEL
LIN {X 0,Y 559.367,Z 536.379,A -85,B 0,C 180,E1 -2773.953,E2 -2773.953} C_VEL
LIN {X 0,Y 559.264,Z 547.23,A -85,B 0,C 180,E1 -2775.838,E2 -2775.838} C_VEL
LIN {X 0,Y 559.841,Z 550.892,A -85,B 0,C 180,E1 -2775.937,E2 -2775.937} C_VEL
LIN {X 0,Y 560.303,Z 554.748,A -85,B 0,C 180,E1 -2775.999,E2 -2775.999} C_VEL
LIN {X 0,Y 560.052,Z 653.973,A -85,B 0,C 180,E1 -2777.291,E2 -2777.291} C_VEL
LIN {X 0,Y 559.922,Z 667.239,A -85,B 0,C 180,E1 -2777.61,E2 -2777.61} C_VEL
LIN {X 0,Y 559.8,Z 679.392,A -85,B 0,C 180,E1 -2778.045,E2 -2778.045} C_VEL
LIN {X 0,Y 559.65,Z 691.071,A -85,B 0,C 180,E1 -2778.606,E2 -2778.606} C_VEL
LIN {X 0,Y 559.486,Z 702.558,A -85,B 0,C 180,E1 -2779.322,E2 -2779.322} C_VEL
LIN {X 0,Y 559.306,Z 713.074,A -85,B 0,C 180,E1 -2780.142,E2 -2780.142} C_VEL
LIN {X 0,Y 559.197,Z 721.671,A -85,B 0,C 180,E1 -2780.961,E2 -2780.961} C_VEL
LIN {X 0,Y 559.051,Z 729.592,A -85,B 0,C 180,E1 -2781.869,E2 -2781.869} C_VEL
LIN {X 0,Y 558.969,Z 737.451,A -85,B 0,C 180,E1 -2782.976,E2 -2782.976} C_VEL
LIN {X 0,Y 558.936,Z 744.452,A -85,B 0,C 180,E1 -2784.226,E2 -2784.226} C_VEL
LIN {X 0,Y 558.826,Z 749.194,A -85,B 0,C 180,E1 -2785.31,E2 -2785.31} C_VEL
LIN {X 0,Y 558.836,Z 752.826,A -85,B 0,C 180,E1 -2786.394,E2 -2786.394} C_VEL
LIN {X 0,Y 558.799,Z 754.703,A -85,B 0,C 180,E1 -2787.116,E2 -2787.116} C_VEL
LIN {X 0,Y 558.746,Z 756.128,A -85,B 0,C 180,E1 -2787.837,E2 -2787.837} C_VEL
LIN {X 0,Y 558.741,Z 757.756,A -85,B 0,C 180,E1 -2789.279,E2 -2789.279} C_VEL
LIN {X 0,Y 558.74,Z 757.996,A -85,B 0,C 180,E1 -2789.999,E2 -2789.999} C_VEL
LIN {X 0,Y 558.741,Z 757.815,A -85,B 0,C 180,E1 -2790.72,E2 -2790.72} C_VEL
LIN {X 0,Y 558.746,Z 756.27,A -85,B 0,C 180,E1 -2792.162,E2 -2792.162} C_VEL
LIN {X 0,Y 558.8,Z 754.909,A -85,B 0,C 180,E1 -2792.883,E2 -2792.883} C_VEL
LIN {X 0,Y 558.844,Z 752.03,A -85,B 0,C 180,E1 -2793.966,E2 -2793.966} C_VEL
LIN {X 0,Y 558.798,Z 748.129,A -85,B 0,C 180,E1 -2795.05,E2 -2795.05} C_VEL
LIN {X 0,Y 558.909,Z 743.097,A -85,B 0,C 180,E1 -2796.135,E2 -2796.135} C_VEL
LIN {X 0,Y 558.972,Z 736.773,A -85,B 0,C 180,E1 -2797.222,E2 -2797.222} C_VEL
LIN {X 0,Y 559.096,Z 728.85,A -85,B 0,C 180,E1 -2798.311,E2 -2798.311} C_VEL
LIN {X 0,Y 559.223,Z 718.998,A -85,B 0,C 180,E1 -2799.402,E2 -2799.402} C_VEL
LIN {X 0,Y 559.416,Z 708.682,A -85,B 0,C 180,E1 -2800.312,E2 -2800.312} C_VEL
LIN {X 0,Y 559.578,Z 697.759,A -85,B 0,C 180,E1 -2801.087,E2 -2801.087} C_VEL
LIN {X 0,Y 559.723,Z 686.187,A -85,B 0,C 180,E1 -2801.738,E2 -2801.738} C_VEL
LIN {X 0,Y 559.881,Z 673.603,A -85,B 0,C 180,E1 -2802.27,E2 -2802.27} C_VEL
LIN {X 0,Y 559.991,Z 660.427,A -85,B 0,C 180,E1 -2802.663,E2 -2802.663} C_VEL
LIN {X 0,Y 560.09,Z 648.058,A -85,B 0,C 180,E1 -2802.892,E2 -2802.892} C_VEL
LIN {X 0,Y 560.168,Z 552.702,A -85,B 0,C 180,E1 -2804.121,E2 -2804.121} C_VEL
LIN {X 0,Y 559.282,Z 547.55,A -85,B 0,C 180,E1 -2804.23,E2 -2804.23} C_VEL
LIN {X 0,Y 559.231,Z 546.34,A -85,B 0,C 180,E1 -2804.37,E2 -2804.37} C_VEL
LIN {X 0,Y 559.443,Z 529.865,A -85,B 0,C 180,E1 -2807.301,E2 -2807.301} C_VEL
LIN {X 0,Y 559.542,Z 517.108,A -85,B 0,C 180,E1 -2809.606,E2 -2809.606} C_VEL
LIN {X 0,Y 559.217,Z 514.889,A -85,B 0,C 180,E1 -2810.074,E2 -2810.074} C_VEL
LIN {X 0,Y 559.133,Z 514.837,A -85,B 0,C 180,E1 -2812.932,E2 -2812.932} C_VEL
LIN {X 0,Y 559.177,Z 514.835,A -85,B 0,C 180,E1 -2815.297,E2 -2815.297} C_VEL
LIN {X 0,Y 559.189,Z 514.829,A -85,B 0,C 180,E1 -2817.711,E2 -2817.711} C_VEL
LIN {X 0,Y 559.156,Z 514.828,A -85,B 0,C 180,E1 -2820.182,E2 -2820.182} C_VEL
LIN {X 0,Y 559.175,Z 514.827,A -85,B 0,C 180,E1 -2822.713,E2 -2822.713} C_VEL
LIN {X 0,Y 559.156,Z 514.838,A -85,B 0,C 180,E1 -2825.321,E2 -2825.321} C_VEL
LIN {X 0,Y 559.134,Z 514.833,A -85,B 0,C 180,E1 -2828.016,E2 -2828.016} C_VEL
LIN {X 0,Y 559.174,Z 514.826,A -85,B 0,C 180,E1 -2830.81,E2 -2830.81} C_VEL
LIN {X 0,Y 559.16,Z 514.831,A -85,B 0,C 180,E1 -2833.731,E2 -2833.731} C_VEL
LIN {X 0,Y 559.142,Z 514.831,A -85,B 0,C 180,E1 -2836.803,E2 -2836.803} C_VEL
LIN {X 0,Y 559.173,Z 514.832,A -85,B 0,C 180,E1 -2839.189,E2 -2839.189} C_VEL
LIN {X 0,Y 559.131,Z 514.831,A -85,B 0,C 180,E1 -2841.982,E2 -2841.982} C_VEL
LIN {X 0,Y 559.154,Z 514.829,A -85,B 0,C 180,E1 -2844.678,E2 -2844.678} C_VEL
LIN {X 0,Y 559.17,Z 514.835,A -85,B 0,C 180,E1 -2847.361,E2 -2847.361} C_VEL
LIN {X 0,Y 559.184,Z 514.826,A -85,B 0,C 180,E1 -2850.134,E2 -2850.134} C_VEL
LIN {X 0,Y 559.177,Z 514.829,A -85,B 0,C 180,E1 -2853.169,E2 -2853.169} C_VEL
LIN {X 0,Y 559.152,Z 514.839,A -85,B 0,C 180,E1 -2855.495,E2 -2855.495} C_VEL
LIN {X 0,Y 559.171,Z 514.825,A -85,B 0,C 180,E1 -2858.624,E2 -2858.624} C_VEL
LIN {X 0,Y 559.166,Z 514.829,A -85,B 0,C 180,E1 -2860.926,E2 -2860.926} C_VEL
LIN {X 0,Y 559.165,Z 514.829,A -85,B 0,C 180,E1 -2863.948,E2 -2863.948} C_VEL
LIN {X 0,Y 559.166,Z 514.828,A -85,B 0,C 180,E1 -2866.184,E2 -2866.184} C_VEL
LIN {X 0,Y 559.189,Z 514.827,A -85,B 0,C 180,E1 -2869.133,E2 -2869.133} C_VEL
LIN {X 0,Y 559.202,Z 514.825,A -85,B 0,C 180,E1 -2872.054,E2 -2872.054} C_VEL
LIN {X 0,Y 559.252,Z 514.818,A -85,B 0,C 180,E1 -2874.953,E2 -2874.953} C_VEL
LIN {X 0,Y 559.245,Z 514.822,A -85,B 0,C 180,E1 -2877.839,E2 -2877.839} C_VEL
LIN {X 0,Y 559.269,Z 514.814,A -85,B 0,C 180,E1 -2880.72,E2 -2880.72} C_VEL
LIN {X 0,Y 559.238,Z 514.818,A -85,B 0,C 180,E1 -2882.881,E2 -2882.881} C_VEL
LIN {X 0,Y 559.222,Z 514.827,A -85,B 0,C 180,E1 -2885.77,E2 -2885.77} C_VEL
LIN {X 0,Y 559.186,Z 514.824,A -85,B 0,C 180,E1 -2888.674,E2 -2888.674} C_VEL
LIN {X 0,Y 559.198,Z 514.832,A -85,B 0,C 180,E1 -2891.601,E2 -2891.601} C_VEL
LIN {X 0,Y 559.192,Z 514.823,A -85,B 0,C 180,E1 -2894.596,E2 -2894.596} C_VEL
LIN {X 0,Y 559.157,Z 514.836,A -85,B 0,C 180,E1 -2897.557,E2 -2897.557} C_VEL
LIN {X 0,Y 559.168,Z 514.833,A -85,B 0,C 180,E1 -2899.838,E2 -2899.838} C_VEL
LIN {X 0,Y 559.136,Z 514.832,A -85,B 0,C 180,E1 -2902.153,E2 -2902.153} C_VEL
LIN {X 0,Y 559.173,Z 514.83,A -85,B 0,C 180,E1 -2905.188,E2 -2905.188} C_VEL
LIN {X 0,Y 559.189,Z 514.833,A -85,B 0,C 180,E1 -2907.712,E2 -2907.712} C_VEL
LIN {X 0,Y 559.157,Z 514.829,A -85,B 0,C 180,E1 -2911.019,E2 -2911.019} C_VEL
LIN {X 0,Y 559.173,Z 514.831,A -85,B 0,C 180,E1 -2913.952,E2 -2913.952} C_VEL
LIN {X 0,Y 559.164,Z 514.824,A -85,B 0,C 180,E1 -2916.449,E2 -2916.449} C_VEL
LIN {X 0,Y 559.173,Z 514.827,A -85,B 0,C 180,E1 -2918.934,E2 -2918.934} C_VEL
LIN {X 0,Y 559.187,Z 514.83,A -85,B 0,C 180,E1 -2921.768,E2 -2921.768} C_VEL
LIN {X 0,Y 559.135,Z 514.831,A -85,B 0,C 180,E1 -2924.74,E2 -2924.74} C_VEL
LIN {X 0,Y 559.165,Z 514.829,A -85,B 0,C 180,E1 -2927.258,E2 -2927.258} C_VEL
LIN {X 0,Y 559.183,Z 514.827,A -85,B 0,C 180,E1 -2930.136,E2 -2930.136} C_VEL
LIN {X 0,Y 559.143,Z 514.827,A -85,B 0,C 180,E1 -2932.893,E2 -2932.893} C_VEL
LIN {X 0,Y 559.164,Z 514.829,A -85,B 0,C 180,E1 -2936.052,E2 -2936.052} C_VEL
LIN {X 0,Y 559.162,Z 514.813,A -85,B 0,C 180,E1 -2938.982,E2 -2938.982} C_VEL
LIN {X 0,Y 559.188,Z 514.826,A -85,B 0,C 180,E1 -2942.289,E2 -2942.289} C_VEL
LIN {X 0,Y 559.179,Z 514.828,A -85,B 0,C 180,E1 -2944.814,E2 -2944.814} C_VEL
LIN {X 0,Y 559.206,Z 515.04,A -85,B 0,C 180,E1 -2946.607,E2 -2946.607} C_VEL
LIN {X 0,Y 560.178,Z 520.515,A -85,B 0,C 180,E1 -2947.503,E2 -2947.503} C_VEL
LIN {X 0,Y 559.838,Z 539.746,A -85,B 0,C 180,E1 -2950.426,E2 -2950.426} C_VEL
LIN {X 0,Y 559.56,Z 558.324,A -85,B 0,C 180,E1 -2953.21,E2 -2953.21} C_VEL
LIN {X 0,Y 559.391,Z 576.037,A -85,B 0,C 180,E1 -2955.796,E2 -2955.796} C_VEL
LIN {X 0,Y 560.307,Z 583.354,A -85,B 0,C 180,E1 -2955.936,E2 -2955.936} C_VEL
LIN {X 0,Y 560.066,Z 683.981,A -85,B 0,C 180,E1 -2957.246,E2 -2957.246} C_VEL
LIN {X 0,Y 559.937,Z 696.474,A -85,B 0,C 180,E1 -2957.543,E2 -2957.543} C_VEL
LIN {X 0,Y 559.818,Z 709.388,A -85,B 0,C 180,E1 -2958,E2 -2958} C_VEL
LIN {X 0,Y 559.667,Z 720.824,A -85,B 0,C 180,E1 -2958.548,E2 -2958.548} C_VEL
LIN {X 0,Y 559.507,Z 731.919,A -85,B 0,C 180,E1 -2959.232,E2 -2959.232} C_VEL
LIN {X 0,Y 559.309,Z 742.548,A -85,B 0,C 180,E1 -2960.051,E2 -2960.051} C_VEL
LIN {X 0,Y 559.161,Z 752.12,A -85,B 0,C 180,E1 -2960.961,E2 -2960.961} C_VEL
LIN {X 0,Y 559.049,Z 759.966,A -85,B 0,C 180,E1 -2961.87,E2 -2961.87} C_VEL
LIN {X 0,Y 558.943,Z 767.627,A -85,B 0,C 180,E1 -2962.959,E2 -2962.959} C_VEL
LIN {X 0,Y 558.935,Z 774.683,A -85,B 0,C 180,E1 -2964.227,E2 -2964.227} C_VEL
LIN {X 0,Y 558.827,Z 779.374,A -85,B 0,C 180,E1 -2965.312,E2 -2965.312} C_VEL
LIN {X 0,Y 558.836,Z 782.961,A -85,B 0,C 180,E1 -2966.395,E2 -2966.395} C_VEL
LIN {X 0,Y 558.799,Z 784.811,A -85,B 0,C 180,E1 -2967.117,E2 -2967.117} C_VEL
LIN {X 0,Y 558.745,Z 787.187,A -85,B 0,C 180,E1 -2968.559,E2 -2968.559} C_VEL
LIN {X 0,Y 558.74,Z 788,A -85,B 0,C 180,E1 -2970.001,E2 -2970.001} C_VEL
LIN {X 0,Y 558.745,Z 787.184,A -85,B 0,C 180,E1 -2971.442,E2 -2971.442} C_VEL
LIN {X 0,Y 558.799,Z 784.807,A -85,B 0,C 180,E1 -2972.884,E2 -2972.884} C_VEL
LIN {X 0,Y 558.844,Z 781.893,A -85,B 0,C 180,E1 -2973.967,E2 -2973.967} C_VEL
LIN {X 0,Y 558.799,Z 777.947,A -85,B 0,C 180,E1 -2975.051,E2 -2975.051} C_VEL
LIN {X 0,Y 558.921,Z 772.864,A -85,B 0,C 180,E1 -2976.136,E2 -2976.136} C_VEL
LIN {X 0,Y 558.978,Z 766.464,A -85,B 0,C 180,E1 -2977.223,E2 -2977.223} C_VEL
LIN {X 0,Y 559.099,Z 758.473,A -85,B 0,C 180,E1 -2978.312,E2 -2978.312} C_VEL
LIN {X 0,Y 559.185,Z 750.329,A -85,B 0,C 180,E1 -2979.222,E2 -2979.222} C_VEL
LIN {X 0,Y 559.34,Z 740.394,A -85,B 0,C 180,E1 -2980.132,E2 -2980.132} C_VEL
LIN {X 0,Y 559.53,Z 729.388,A -85,B 0,C 180,E1 -2980.938,E2 -2980.938} C_VEL
LIN {X 0,Y 559.673,Z 717.451,A -85,B 0,C 180,E1 -2981.628,E2 -2981.628} C_VEL
LIN {X 0,Y 559.842,Z 704.76,A -85,B 0,C 180,E1 -2982.185,E2 -2982.185} C_VEL
LIN {X 0,Y 559.998,Z 691.331,A -85,B 0,C 180,E1 -2982.595,E2 -2982.595} C_VEL
LIN {X 0,Y 560.087,Z 678.046,A -85,B 0,C 180,E1 -2982.847,E2 -2982.847} C_VEL
LIN {X 0,Y 560.191,Z 581.367,A -85,B 0,C 180,E1 -2984.093,E2 -2984.093} C_VEL
LIN {X 0,Y 559.395,Z 576.018,A -85,B 0,C 180,E1 -2984.205,E2 -2984.205} C_VEL
LIN {X 0,Y 559.606,Z 556.4,A -85,B 0,C 180,E1 -2987.076,E2 -2987.076} C_VEL
LIN {X 0,Y 559.918,Z 536.907,A -85,B 0,C 180,E1 -2990.002,E2 -2990.002} C_VEL
LIN {X 0,Y 560.149,Z 520.503,A -85,B 0,C 180,E1 -2992.5,E2 -2992.5} C_VEL
LIN {X 0,Y 559.157,Z 514.916,A -85,B 0,C 180,E1 -2993.432,E2 -2993.432} C_VEL
LIN {X 0,Y 559.183,Z 514.829,A -85,B 0,C 180,E1 -2996.097,E2 -2996.097} C_VEL
LIN {X 0,Y 559.167,Z 514.829,A -85,B 0,C 180,E1 -2998.53,E2 -2998.53} C_VEL
LIN {X 0,Y 559.15,Z 514.83,A -85,B 0,C 180,E1 -3001.273,E2 -3001.273} C_VEL
LIN {X 0,Y 559.17,Z 514.832,A -85,B 0,C 180,E1 -3003.949,E2 -3003.949} C_VEL
LIN {X 0,Y 559.144,Z 514.831,A -85,B 0,C 180,E1 -3007.109,E2 -3007.109} C_VEL
LIN {X 0,Y 559.164,Z 514.833,A -85,B 0,C 180,E1 -3009.942,E2 -3009.942} C_VEL
LIN {X 0,Y 559.167,Z 514.83,A -85,B 0,C 180,E1 -3012.743,E2 -3012.743} C_VEL
LIN {X 0,Y 559.152,Z 514.833,A -85,B 0,C 180,E1 -3015.761,E2 -3015.761} C_VEL
LIN {X 0,Y 559.165,Z 514.837,A -85,B 0,C 180,E1 -3018.23,E2 -3018.23} C_VEL
LIN {X 0,Y 559.179,Z 514.826,A -85,B 0,C 180,E1 -3021.192,E2 -3021.192} C_VEL
LIN {X 0,Y 559.161,Z 514.832,A -85,B 0,C 180,E1 -3023.791,E2 -3023.791} C_VEL
LIN {X 0,Y 559.166,Z 514.835,A -85,B 0,C 180,E1 -3026.425,E2 -3026.425} C_VEL
LIN {X 0,Y 559.158,Z 514.83,A -85,B 0,C 180,E1 -3028.981,E2 -3028.981} C_VEL
LIN {X 0,Y 559.172,Z 514.83,A -85,B 0,C 180,E1 -3031.619,E2 -3031.619} C_VEL
LIN {X 0,Y 559.185,Z 514.833,A -85,B 0,C 180,E1 -3033.903,E2 -3033.903} C_VEL
LIN {X 0,Y 559.209,Z 515.01,A -85,B 0,C 180,E1 -3035.024,E2 -3035.024} C_VEL
LIN {X 0,Y 560.389,Z 521.613,A -85,B 0,C 180,E1 -3035.947,E2 -3035.947} C_VEL
LIN {X 0,Y 560.186,Z 540.383,A -85,B 0,C 180,E1 -3038.483,E2 -3038.483} C_VEL
LIN {X 0,Y 559.868,Z 559.447,A -85,B 0,C 180,E1 -3041.141,E2 -3041.141} C_VEL
LIN {X 0,Y 559.579,Z 579.966,A -85,B 0,C 180,E1 -3043.96,E2 -3043.96} C_VEL
LIN {X 0,Y 559.348,Z 599.118,A -85,B 0,C 180,E1 -3046.559,E2 -3046.559} C_VEL
LIN {X 0,Y 559.188,Z 616.478,A -85,B 0,C 180,E1 -3048.86,E2 -3048.86} C_VEL
LIN {X 0,Y 559.749,Z 622.525,A -85,B 0,C 180,E1 -3048.966,E2 -3048.966} C_VEL
LIN {X 0,Y 559.612,Z 695.763,A -85,B 0,C 180,E1 -3049.919,E2 -3049.919} C_VEL
LIN {X 0,Y 559.526,Z 707.491,A -85,B 0,C 180,E1 -3050.214,E2 -3050.214} C_VEL
LIN {X 0,Y 559.421,Z 717.61,A -85,B 0,C 180,E1 -3050.6,E2 -3050.6} C_VEL
LIN {X 0,Y 559.309,Z 728.045,A -85,B 0,C 180,E1 -3051.145,E2 -3051.145} C_VEL
LIN {X 0,Y 559.179,Z 737.453,A -85,B 0,C 180,E1 -3051.78,E2 -3051.78} C_VEL
LIN {X 0,Y 559.073,Z 746.877,A -85,B 0,C 180,E1 -3052.597,E2 -3052.597} C_VEL
LIN {X 0,Y 558.995,Z 755.045,A -85,B 0,C 180,E1 -3053.503,E2 -3053.503} C_VEL
LIN {X 0,Y 558.926,Z 761.539,A -85,B 0,C 180,E1 -3054.408,E2 -3054.408} C_VEL
LIN {X 0,Y 558.898,Z 766.711,A -85,B 0,C 180,E1 -3055.312,E2 -3055.312} C_VEL
LIN {X 0,Y 558.843,Z 771.457,A -85,B 0,C 180,E1 -3056.395,E2 -3056.395} C_VEL
LIN {X 0,Y 558.806,Z 773.824,A -85,B 0,C 180,E1 -3057.116,E2 -3057.116} C_VEL
LIN {X 0,Y 558.745,Z 775.613,A -85,B 0,C 180,E1 -3057.837,E2 -3057.837} C_VEL
LIN {X 0,Y 558.743,Z 776.913,A -85,B 0,C 180,E1 -3058.559,E2 -3058.559} C_VEL
LIN {X 0,Y 558.738,Z 777.712,A -85,B 0,C 180,E1 -3059.279,E2 -3059.279} C_VEL
LIN {X 0,Y 558.738,Z 777.996,A -85,B 0,C 180,E1 -3060,E2 -3060} C_VEL
LIN {X 0,Y 558.739,Z 777.768,A -85,B 0,C 180,E1 -3060.721,E2 -3060.721} C_VEL
LIN {X 0,Y 558.746,Z 777.032,A -85,B 0,C 180,E1 -3061.442,E2 -3061.442} C_VEL
LIN {X 0,Y 558.747,Z 775.804,A -85,B 0,C 180,E1 -3062.163,E2 -3062.163} C_VEL
LIN {X 0,Y 558.838,Z 772.974,A -85,B 0,C 180,E1 -3063.244,E2 -3063.244} C_VEL
LIN {X 0,Y 558.893,Z 768.86,A -85,B 0,C 180,E1 -3064.327,E2 -3064.327} C_VEL
LIN {X 0,Y 558.881,Z 763.245,A -85,B 0,C 180,E1 -3065.412,E2 -3065.412} C_VEL
LIN {X 0,Y 558.996,Z 757.18,A -85,B 0,C 180,E1 -3066.316,E2 -3066.316} C_VEL
LIN {X 0,Y 559.057,Z 749.523,A -85,B 0,C 180,E1 -3067.222,E2 -3067.222} C_VEL
LIN {X 0,Y 559.157,Z 740.875,A -85,B 0,C 180,E1 -3068.038,E2 -3068.038} C_VEL
LIN {X 0,Y 559.33,Z 730.993,A -85,B 0,C 180,E1 -3068.763,E2 -3068.763} C_VEL
LIN {X 0,Y 559.399,Z 721.412,A -85,B 0,C 180,E1 -3069.309,E2 -3069.309} C_VEL
LIN {X 0,Y 559.518,Z 710.785,A -85,B 0,C 180,E1 -3069.763,E2 -3069.763} C_VEL
LIN {X 0,Y 559.572,Z 699.126,A -85,B 0,C 180,E1 -3070.104,E2 -3070.104} C_VEL
LIN {X 0,Y 559.648,Z 684.63,A -85,B 0,C 180,E1 -3070.332,E2 -3070.332} C_VEL
LIN {X 0,Y 559.625,Z 619.797,A -85,B 0,C 180,E1 -3071.161,E2 -3071.161} C_VEL
LIN {X 0,Y 559.187,Z 616.263,A -85,B 0,C 180,E1 -3071.244,E2 -3071.244} C_VEL
LIN {X 0,Y 559.437,Z 594.309,A -85,B 0,C 180,E1 -3074.18,E2 -3074.18} C_VEL
LIN {X 0,Y 559.65,Z 574.533,A -85,B 0,C 180,E1 -3076.873,E2 -3076.873} C_VEL
LIN {X 0,Y 559.073,Z 571.108,A -85,B 0,C 180,E1 -3077.362,E2 -3077.362} C_VEL
LIN {X 0,Y 553.529,Z 560.635,A -85,B 0,C 180,E1 -3079.007,E2 -3079.007} C_VEL
LIN {X 0,Y 552.992,Z 557.228,A -85,B 0,C 180,E1 -3079.506,E2 -3079.506} C_VEL
LIN {X 0,Y 553.32,Z 536.37,A -85,B 0,C 180,E1 -3082.399,E2 -3082.399} C_VEL
LIN {X 0,Y 553.41,Z 522.122,A -85,B 0,C 180,E1 -3084.377,E2 -3084.377} C_VEL
LIN {X 0,Y 552.166,Z 515.777,A -85,B 0,C 180,E1 -3085.352,E2 -3085.352} C_VEL
LIN {X 0,Y 552.124,Z 515.712,A -85,B 0,C 180,E1 -3088.098,E2 -3088.098} C_VEL
LIN {X 0,Y 552.105,Z 515.709,A -85,B 0,C 180,E1 -3090.609,E2 -3090.609} C_VEL
LIN {X 0,Y 552.119,Z 515.709,A -85,B 0,C 180,E1 -3093.186,E2 -3093.186} C_VEL
LIN {X 0,Y 552.103,Z 515.713,A -85,B 0,C 180,E1 -3095.843,E2 -3095.843} C_VEL
LIN {X 0,Y 552.128,Z 515.707,A -85,B 0,C 180,E1 -3099.062,E2 -3099.062} C_VEL
LIN {X 0,Y 552.124,Z 515.704,A -85,B 0,C 180,E1 -3101.446,E2 -3101.446} C_VEL
LIN {X 0,Y 552.095,Z 515.706,A -85,B 0,C 180,E1 -3104.531,E2 -3104.531} C_VEL
LIN {X 0,Y 552.134,Z 515.708,A -85,B 0,C 180,E1 -3107.585,E2 -3107.585} C_VEL
LIN {X 0,Y 552.134,Z 515.697,A -85,B 0,C 180,E1 -3110.473,E2 -3110.473} C_VEL
LIN {X 0,Y 552.111,Z 515.714,A -85,B 0,C 180,E1 -3113.317,E2 -3113.317} C_VEL
LIN {X 0,Y 552.108,Z 515.706,A -85,B 0,C 180,E1 -3115.937,E2 -3115.937} C_VEL
LIN {X 0,Y 552.124,Z 515.708,A -85,B 0,C 180,E1 -3118.54,E2 -3118.54} C_VEL
LIN {X 0,Y 552.129,Z 515.708,A -85,B 0,C 180,E1 -3121.438,E2 -3121.438} C_VEL
LIN {X 0,Y 552.134,Z 515.707,A -85,B 0,C 180,E1 -3124.355,E2 -3124.355} C_VEL
LIN {X 0,Y 552.101,Z 515.715,A -85,B 0,C 180,E1 -3126.757,E2 -3126.757} C_VEL
LIN {X 0,Y 552.127,Z 515.712,A -85,B 0,C 180,E1 -3129.12,E2 -3129.12} C_VEL
LIN {X 0,Y 552.184,Z 515.887,A -85,B 0,C 180,E1 -3129.961,E2 -3129.961} C_VEL
LIN {X 0,Y 552.59,Z 520.659,A -85,B 0,C 180,E1 -3130.883,E2 -3130.883} C_VEL
LIN {X 0,Y 552.37,Z 535.334,A -85,B 0,C 180,E1 -3133.555,E2 -3133.555} C_VEL
LIN {X 0,Y 552.232,Z 547.196,A -85,B 0,C 180,E1 -3135.65,E2 -3135.65} C_VEL
LIN {X 0,Y 552.733,Z 550.377,A -85,B 0,C 180,E1 -3135.745,E2 -3135.745} C_VEL
LIN {X 0,Y 553.434,Z 555.046,A -85,B 0,C 180,E1 -3135.825,E2 -3135.825} C_VEL
LIN {X 0,Y 553.15,Z 654.002,A -85,B 0,C 180,E1 -3137.129,E2 -3137.129} C_VEL
LIN {X 0,Y 552.989,Z 667.258,A -85,B 0,C 180,E1 -3137.452,E2 -3137.452} C_VEL
LIN {X 0,Y 552.851,Z 679.399,A -85,B 0,C 180,E1 -3137.892,E2 -3137.892} C_VEL
LIN {X 0,Y 552.689,Z 690.893,A -85,B 0,C 180,E1 -3138.45,E2 -3138.45} C_VEL
LIN {X 0,Y 552.51,Z 702.565,A -85,B 0,C 180,E1 -3139.185,E2 -3139.185} C_VEL
LIN {X 0,Y 552.302,Z 713.082,A -85,B 0,C 180,E1 -3140.015,E2 -3140.015} C_VEL
LIN {X 0,Y 552.153,Z 721.677,A -85,B 0,C 180,E1 -3140.845,E2 -3140.845} C_VEL
LIN {X 0,Y 552.008,Z 729.596,A -85,B 0,C 180,E1 -3141.765,E2 -3141.765} C_VEL
LIN {X 0,Y 551.893,Z 737.455,A -85,B 0,C 180,E1 -3142.886,E2 -3142.886} C_VEL
LIN {X 0,Y 551.868,Z 744.455,A -85,B 0,C 180,E1 -3144.152,E2 -3144.152} C_VEL
LIN {X 0,Y 551.725,Z 749.196,A -85,B 0,C 180,E1 -3145.25,E2 -3145.25} C_VEL
LIN {X 0,Y 551.751,Z 752.828,A -85,B 0,C 180,E1 -3146.348,E2 -3146.348} C_VEL
LIN {X 0,Y 551.723,Z 754.705,A -85,B 0,C 180,E1 -3147.079,E2 -3147.079} C_VEL
LIN {X 0,Y 551.656,Z 756.129,A -85,B 0,C 180,E1 -3147.809,E2 -3147.809} C_VEL
LIN {X 0,Y 551.642,Z 757.757,A -85,B 0,C 180,E1 -3149.269,E2 -3149.269} C_VEL
LIN {X 0,Y 551.641,Z 757.996,A -85,B 0,C 180,E1 -3149.999,E2 -3149.999} C_VEL
LIN {X 0,Y 551.641,Z 757.815,A -85,B 0,C 180,E1 -3150.729,E2 -3150.729} C_VEL
LIN {X 0,Y 551.657,Z 756.269,A -85,B 0,C 180,E1 -3152.19,E2 -3152.19} C_VEL
LIN {X 0,Y 551.724,Z 754.908,A -85,B 0,C 180,E1 -3152.92,E2 -3152.92} C_VEL
LIN {X 0,Y 551.764,Z 752.028,A -85,B 0,C 180,E1 -3154.017,E2 -3154.017} C_VEL
LIN {X 0,Y 551.723,Z 748.127,A -85,B 0,C 180,E1 -3155.115,E2 -3155.115} C_VEL
LIN {X 0,Y 551.81,Z 742.398,A -85,B 0,C 180,E1 -3156.348,E2 -3156.348} C_VEL
LIN {X 0,Y 551.924,Z 735.542,A -85,B 0,C 180,E1 -3157.499,E2 -3157.499} C_VEL
LIN {X 0,Y 552.077,Z 727.358,A -85,B 0,C 180,E1 -3158.602,E2 -3158.602} C_VEL
LIN {X 0,Y 552.196,Z 718.992,A -85,B 0,C 180,E1 -3159.523,E2 -3159.523} C_VEL
LIN {X 0,Y 552.409,Z 708.676,A -85,B 0,C 180,E1 -3160.444,E2 -3160.444} C_VEL
LIN {X 0,Y 552.596,Z 698.044,A -85,B 0,C 180,E1 -3161.209,E2 -3161.209} C_VEL
LIN {X 0,Y 552.743,Z 687.274,A -85,B 0,C 180,E1 -3161.83,E2 -3161.83} C_VEL
LIN {X 0,Y 552.92,Z 674.753,A -85,B 0,C 180,E1 -3162.385,E2 -3162.385} C_VEL
LIN {X 0,Y 553.051,Z 661.321,A -85,B 0,C 180,E1 -3162.802,E2 -3162.802} C_VEL
LIN {X 0,Y 553.193,Z 648.017,A -85,B 0,C 180,E1 -3163.055,E2 -3163.055} C_VEL
LIN {X 0,Y 553.332,Z 553.686,A -85,B 0,C 180,E1 -3164.286,E2 -3164.286} C_VEL
LIN {X 0,Y 552.259,Z 547.491,A -85,B 0,C 180,E1 -3164.418,E2 -3164.418} C_VEL
LIN {X 0,Y 552.22,Z 545.276,A -85,B 0,C 180,E1 -3164.745,E2 -3164.745} C_VEL
LIN {X 0,Y 552.428,Z 530.477,A -85,B 0,C 180,E1 -3167.416,E2 -3167.416} C_VEL
LIN {X 0,Y 552.579,Z 518.47,A -85,B 0,C 180,E1 -3169.615,E2 -3169.615} C_VEL
LIN {X 0,Y 552.178,Z 515.759,A -85,B 0,C 180,E1 -3170.196,E2 -3170.196} C_VEL
LIN {X 0,Y 552.112,Z 515.715,A -85,B 0,C 180,E1 -3173.241,E2 -3173.241} C_VEL
LIN {X 0,Y 552.131,Z 515.708,A -85,B 0,C 180,E1 -3175.643,E2 -3175.643} C_VEL
LIN {X 0,Y 552.124,Z 515.705,A -85,B 0,C 180,E1 -3178.561,E2 -3178.561} C_VEL
LIN {X 0,Y 552.135,Z 515.712,A -85,B 0,C 180,E1 -3181.479,E2 -3181.479} C_VEL
LIN {X 0,Y 552.136,Z 515.704,A -85,B 0,C 180,E1 -3184.17,E2 -3184.17} C_VEL
LIN {X 0,Y 552.11,Z 515.706,A -85,B 0,C 180,E1 -3186.746,E2 -3186.746} C_VEL
LIN {X 0,Y 552.132,Z 515.71,A -85,B 0,C 180,E1 -3189.526,E2 -3189.526} C_VEL
LIN {X 0,Y 552.128,Z 515.704,A -85,B 0,C 180,E1 -3192.424,E2 -3192.424} C_VEL
LIN {X 0,Y 552.094,Z 515.715,A -85,B 0,C 180,E1 -3195.562,E2 -3195.562} C_VEL
LIN {X 0,Y 552.136,Z 515.703,A -85,B 0,C 180,E1 -3198.675,E2 -3198.675} C_VEL
LIN {X 0,Y 552.116,Z 515.71,A -85,B 0,C 180,E1 -3201.411,E2 -3201.411} C_VEL
LIN {X 0,Y 552.109,Z 515.707,A -85,B 0,C 180,E1 -3204.158,E2 -3204.158} C_VEL
LIN {X 0,Y 552.124,Z 515.705,A -85,B 0,C 180,E1 -3206.815,E2 -3206.815} C_VEL
LIN {X 0,Y 552.109,Z 515.714,A -85,B 0,C 180,E1 -3209.391,E2 -3209.391} C_VEL
LIN {X 0,Y 552.122,Z 515.706,A -85,B 0,C 180,E1 -3211.902,E2 -3211.902} C_VEL
LIN {X 0,Y 552.151,Z 515.701,A -85,B 0,C 180,E1 -3214.649,E2 -3214.649} C_VEL
LIN {X 0,Y 552.09,Z 515.716,A -85,B 0,C 180,E1 -3217.549,E2 -3217.549} C_VEL
LIN {X 0,Y 552.143,Z 515.702,A -85,B 0,C 180,E1 -3220.373,E2 -3220.373} C_VEL
LIN {X 0,Y 552.151,Z 515.702,A -85,B 0,C 180,E1 -3222.977,E2 -3222.977} C_VEL
LIN {X 0,Y 552.129,Z 515.706,A -85,B 0,C 180,E1 -3226.004,E2 -3226.004} C_VEL
LIN {X 0,Y 552.156,Z 515.702,A -85,B 0,C 180,E1 -3228.993,E2 -3228.993} C_VEL
LIN {X 0,Y 552.156,Z 515.704,A -85,B 0,C 180,E1 -3231.951,E2 -3231.951} C_VEL
LIN {X 0,Y 552.226,Z 515.693,A -85,B 0,C 180,E1 -3234.889,E2 -3234.889} C_VEL
LIN {X 0,Y 552.217,Z 515.698,A -85,B 0,C 180,E1 -3237.812,E2 -3237.812} C_VEL
LIN {X 0,Y 552.239,Z 515.69,A -85,B 0,C 180,E1 -3240.729,E2 -3240.729} C_VEL
LIN {X 0,Y 552.204,Z 515.694,A -85,B 0,C 180,E1 -3242.918,E2 -3242.918} C_VEL
LIN {X 0,Y 552.192,Z 515.701,A -85,B 0,C 180,E1 -3245.844,E2 -3245.844} C_VEL
LIN {X 0,Y 552.156,Z 515.7,A -85,B 0,C 180,E1 -3248.786,E2 -3248.786} C_VEL
LIN {X 0,Y 552.155,Z 515.708,A -85,B 0,C 180,E1 -3251.751,E2 -3251.751} C_VEL
LIN {X 0,Y 552.129,Z 515.703,A -85,B 0,C 180,E1 -3254.749,E2 -3254.749} C_VEL
LIN {X 0,Y 552.108,Z 515.713,A -85,B 0,C 180,E1 -3257.789,E2 -3257.789} C_VEL
LIN {X 0,Y 552.127,Z 515.706,A -85,B 0,C 180,E1 -3260.101,E2 -3260.101} C_VEL
LIN {X 0,Y 552.089,Z 515.708,A -85,B 0,C 180,E1 -3262.451,E2 -3262.451} C_VEL
LIN {X 0,Y 552.151,Z 515.707,A -85,B 0,C 180,E1 -3265.351,E2 -3265.351} C_VEL
LIN {X 0,Y 552.12,Z 515.708,A -85,B 0,C 180,E1 -3268.098,E2 -3268.098} C_VEL
LIN {X 0,Y 552.101,Z 515.706,A -85,B 0,C 180,E1 -3270.609,E2 -3270.609} C_VEL
LIN {X 0,Y 552.124,Z 515.707,A -85,B 0,C 180,E1 -3273.185,E2 -3273.185} C_VEL
LIN {X 0,Y 552.109,Z 515.709,A -85,B 0,C 180,E1 -3275.842,E2 -3275.842} C_VEL
LIN {X 0,Y 552.121,Z 515.706,A -85,B 0,C 180,E1 -3279.063,E2 -3279.063} C_VEL
LIN {X 0,Y 552.135,Z 515.709,A -85,B 0,C 180,E1 -3281.445,E2 -3281.445} C_VEL
LIN {X 0,Y 552.091,Z 515.709,A -85,B 0,C 180,E1 -3284.533,E2 -3284.533} C_VEL
LIN {X 0,Y 552.128,Z 515.711,A -85,B 0,C 180,E1 -3287.585,E2 -3287.585} C_VEL
LIN {X 0,Y 552.131,Z 515.702,A -85,B 0,C 180,E1 -3290.474,E2 -3290.474} C_VEL
LIN {X 0,Y 552.11,Z 515.706,A -85,B 0,C 180,E1 -3293.317,E2 -3293.317} C_VEL
LIN {X 0,Y 552.127,Z 515.708,A -85,B 0,C 180,E1 -3295.94,E2 -3295.94} C_VEL
LIN {X 0,Y 552.117,Z 515.689,A -85,B 0,C 180,E1 -3298.541,E2 -3298.541} C_VEL
LIN {X 0,Y 552.123,Z 515.71,A -85,B 0,C 180,E1 -3301.439,E2 -3301.439} C_VEL
LIN {X 0,Y 552.13,Z 515.702,A -85,B 0,C 180,E1 -3304.357,E2 -3304.357} C_VEL
LIN {X 0,Y 552.146,Z 515.888,A -85,B 0,C 180,E1 -3306.448,E2 -3306.448} C_VEL
LIN {X 0,Y 553.221,Z 521.628,A -85,B 0,C 180,E1 -3307.401,E2 -3307.401} C_VEL
LIN {X 0,Y 552.899,Z 541.412,A -85,B 0,C 180,E1 -3310.426,E2 -3310.426} C_VEL
LIN {X 0,Y 552.569,Z 559.584,A -85,B 0,C 180,E1 -3313.182,E2 -3313.182} C_VEL
LIN {X 0,Y 552.393,Z 575.99,A -85,B 0,C 180,E1 -3315.609,E2 -3315.609} C_VEL
LIN {X 0,Y 553.434,Z 583.828,A -85,B 0,C 180,E1 -3315.764,E2 -3315.764} C_VEL
LIN {X 0,Y 553.157,Z 683.981,A -85,B 0,C 180,E1 -3317.084,E2 -3317.084} C_VEL
LIN {X 0,Y 553.012,Z 697.234,A -85,B 0,C 180,E1 -3317.407,E2 -3317.407} C_VEL
LIN {X 0,Y 552.857,Z 709.381,A -85,B 0,C 180,E1 -3317.846,E2 -3317.846} C_VEL
LIN {X 0,Y 552.689,Z 721.676,A -85,B 0,C 180,E1 -3318.45,E2 -3318.45} C_VEL
LIN {X 0,Y 552.505,Z 733.208,A -85,B 0,C 180,E1 -3319.187,E2 -3319.187} C_VEL
LIN {X 0,Y 552.295,Z 743.611,A -85,B 0,C 180,E1 -3320.016,E2 -3320.016} C_VEL
LIN {X 0,Y 552.125,Z 752.12,A -85,B 0,C 180,E1 -3320.845,E2 -3320.845} C_VEL
LIN {X 0,Y 552.012,Z 759.966,A -85,B 0,C 180,E1 -3321.766,E2 -3321.766} C_VEL
LIN {X 0,Y 551.889,Z 767.626,A -85,B 0,C 180,E1 -3322.868,E2 -3322.868} C_VEL
LIN {X 0,Y 551.867,Z 774.682,A -85,B 0,C 180,E1 -3324.153,E2 -3324.153} C_VEL
LIN {X 0,Y 551.725,Z 779.374,A -85,B 0,C 180,E1 -3325.251,E2 -3325.251} C_VEL
LIN {X 0,Y 551.75,Z 782.962,A -85,B 0,C 180,E1 -3326.349,E2 -3326.349} C_VEL
LIN {X 0,Y 551.723,Z 784.811,A -85,B 0,C 180,E1 -3327.08,E2 -3327.08} C_VEL
LIN {X 0,Y 551.645,Z 787.186,A -85,B 0,C 180,E1 -3328.541,E2 -3328.541} C_VEL
LIN {X 0,Y 551.64,Z 788,A -85,B 0,C 180,E1 -3330.001,E2 -3330.001} C_VEL
LIN {X 0,Y 551.645,Z 787.184,A -85,B 0,C 180,E1 -3331.461,E2 -3331.461} C_VEL
LIN {X 0,Y 551.724,Z 784.806,A -85,B 0,C 180,E1 -3332.921,E2 -3332.921} C_VEL
LIN {X 0,Y 551.764,Z 781.893,A -85,B 0,C 180,E1 -3334.018,E2 -3334.018} C_VEL
LIN {X 0,Y 551.724,Z 777.947,A -85,B 0,C 180,E1 -3335.116,E2 -3335.116} C_VEL
LIN {X 0,Y 551.803,Z 772.189,A -85,B 0,C 180,E1 -3336.342,E2 -3336.342} C_VEL
LIN {X 0,Y 551.927,Z 765.233,A -85,B 0,C 180,E1 -3337.5,E2 -3337.5} C_VEL
LIN {X 0,Y 552.083,Z 756.987,A -85,B 0,C 180,E1 -3338.603,E2 -3338.603} C_VEL
LIN {X 0,Y 552.222,Z 748.533,A -85,B 0,C 180,E1 -3339.524,E2 -3339.524} C_VEL
LIN {X 0,Y 552.385,Z 738.089,A -85,B 0,C 180,E1 -3340.446,E2 -3340.446} C_VEL
LIN {X 0,Y 552.6,Z 727.278,A -85,B 0,C 180,E1 -3341.214,E2 -3341.214} C_VEL
LIN {X 0,Y 552.754,Z 716.399,A -85,B 0,C 180,E1 -3341.831,E2 -3341.831} C_VEL
LIN {X 0,Y 552.908,Z 704.757,A -85,B 0,C 180,E1 -3342.34,E2 -3342.34} C_VEL
LIN {X 0,Y 553.057,Z 691.331,A -85,B 0,C 180,E1 -3342.756,E2 -3342.756} C_VEL
LIN {X 0,Y 553.19,Z 678.046,A -85,B 0,C 180,E1 -3343.01,E2 -3343.01} C_VEL
LIN {X 0,Y 553.403,Z 582.64,A -85,B 0,C 180,E1 -3344.253,E2 -3344.253} C_VEL
LIN {X 0,Y 552.405,Z 575.972,A -85,B 0,C 180,E1 -3344.392,E2 -3344.392} C_VEL
LIN {X 0,Y 552.667,Z 555.091,A -85,B 0,C 180,E1 -3347.495,E2 -3347.495} C_VEL
LIN {X 0,Y 553.023,Z 534.355,A -85,B 0,C 180,E1 -3350.65,E2 -3350.65} C_VEL
LIN {X 0,Y 553.19,Z 521.605,A -85,B 0,C 180,E1 -3352.601,E2 -3352.601} C_VEL
LIN {X 0,Y 552.127,Z 515.829,A -85,B 0,C 180,E1 -3353.582,E2 -3353.582} C_VEL
LIN {X 0,Y 552.133,Z 515.704,A -85,B 0,C 180,E1 -3355.645,E2 -3355.645} C_VEL
LIN {X 0,Y 552.129,Z 515.705,A -85,B 0,C 180,E1 -3358.562,E2 -3358.562} C_VEL
LIN {X 0,Y 552.115,Z 515.707,A -85,B 0,C 180,E1 -3361.476,E2 -3361.476} C_VEL
LIN {X 0,Y 552.137,Z 515.712,A -85,B 0,C 180,E1 -3364.17,E2 -3364.17} C_VEL
LIN {X 0,Y 552.109,Z 515.709,A -85,B 0,C 180,E1 -3366.747,E2 -3366.747} C_VEL
LIN {X 0,Y 552.133,Z 515.705,A -85,B 0,C 180,E1 -3369.527,E2 -3369.527} C_VEL
LIN {X 0,Y 552.135,Z 515.711,A -85,B 0,C 180,E1 -3372.425,E2 -3372.425} C_VEL
LIN {X 0,Y 552.097,Z 515.71,A -85,B 0,C 180,E1 -3375.562,E2 -3375.562} C_VEL
LIN {X 0,Y 552.124,Z 515.71,A -85,B 0,C 180,E1 -3378.554,E2 -3378.554} C_VEL
LIN {X 0,Y 552.122,Z 515.706,A -85,B 0,C 180,E1 -3381.411,E2 -3381.411} C_VEL
LIN {X 0,Y 552.104,Z 515.716,A -85,B 0,C 180,E1 -3384.158,E2 -3384.158} C_VEL
LIN {X 0,Y 552.119,Z 515.708,A -85,B 0,C 180,E1 -3386.814,E2 -3386.814} C_VEL
LIN {X 0,Y 552.105,Z 515.709,A -85,B 0,C 180,E1 -3389.391,E2 -3389.391} C_VEL
LIN {X 0,Y 552.127,Z 515.712,A -85,B 0,C 180,E1 -3391.903,E2 -3391.903} C_VEL
LIN {X 0,Y 552.179,Z 515.858,A -85,B 0,C 180,E1 -3394.934,E2 -3394.934} C_VEL
LIN {X 0,Y 553.35,Z 522.15,A -85,B 0,C 180,E1 -3395.82,E2 -3395.82} C_VEL
LIN {X 0,Y 553.217,Z 539.28,A -85,B 0,C 180,E1 -3398.125,E2 -3398.125} C_VEL
LIN {X 0,Y 553.015,Z 557.034,A -85,B 0,C 180,E1 -3400.557,E2 -3400.557} C_VEL
LIN {X 0,Y 552.636,Z 577.235,A -85,B 0,C 180,E1 -3403.373,E2 -3403.373} C_VEL
LIN {X 0,Y 552.355,Z 597.755,A -85,B 0,C 180,E1 -3406.198,E2 -3406.198} C_VEL
LIN {X 0,Y 552.159,Z 616.29,A -85,B 0,C 180,E1 -3408.703,E2 -3408.703} C_VEL
LIN {X 0,Y 552.781,Z 622.342,A -85,B 0,C 180,E1 -3408.822,E2 -3408.822} C_VEL
LIN {X 0,Y 552.648,Z 695.796,A -85,B 0,C 180,E1 -3409.791,E2 -3409.791} C_VEL
LIN {X 0,Y 552.539,Z 707.5,A -85,B 0,C 180,E1 -3410.089,E2 -3410.089} C_VEL
LIN {X 0,Y 552.428,Z 717.62,A -85,B 0,C 180,E1 -3410.48,E2 -3410.48} C_VEL
LIN {X 0,Y 552.289,Z 728.063,A -85,B 0,C 180,E1 -3411.032,E2 -3411.032} C_VEL
LIN {X 0,Y 552.143,Z 737.467,A -85,B 0,C 180,E1 -3411.675,E2 -3411.675} C_VEL
LIN {X 0,Y 552.011,Z 746.88,A -85,B 0,C 180,E1 -3412.502,E2 -3412.502} C_VEL
LIN {X 0,Y 551.93,Z 755.051,A -85,B 0,C 180,E1 -3413.419,E2 -3413.419} C_VEL
LIN {X 0,Y 551.87,Z 761.545,A -85,B 0,C 180,E1 -3414.336,E2 -3414.336} C_VEL
LIN {X 0,Y 551.807,Z 766.72,A -85,B 0,C 180,E1 -3415.251,E2 -3415.251} C_VEL
LIN {X 0,Y 551.758,Z 771.459,A -85,B 0,C 180,E1 -3416.349,E2 -3416.349} C_VEL
LIN {X 0,Y 551.732,Z 773.825,A -85,B 0,C 180,E1 -3417.079,E2 -3417.079} C_VEL
LIN {X 0,Y 551.656,Z 775.616,A -85,B 0,C 180,E1 -3417.81,E2 -3417.81} C_VEL
LIN {X 0,Y 551.642,Z 776.913,A -85,B 0,C 180,E1 -3418.54,E2 -3418.54} C_VEL
LIN {X 0,Y 551.638,Z 777.711,A -85,B 0,C 180,E1 -3419.27,E2 -3419.27} C_VEL
LIN {X 0,Y 551.638,Z 777.996,A -85,B 0,C 180,E1 -3420,E2 -3420} C_VEL
LIN {X 0,Y 551.64,Z 777.772,A -85,B 0,C 180,E1 -3420.73,E2 -3420.73} C_VEL
LIN {X 0,Y 551.646,Z 777.037,A -85,B 0,C 180,E1 -3421.46,E2 -3421.46} C_VEL
LIN {X 0,Y 551.657,Z 775.804,A -85,B 0,C 180,E1 -3422.19,E2 -3422.19} C_VEL
LIN {X 0,Y 551.763,Z 772.978,A -85,B 0,C 180,E1 -3423.286,E2 -3423.286} C_VEL
LIN {X 0,Y 551.806,Z 768.862,A -85,B 0,C 180,E1 -3424.383,E2 -3424.383} C_VEL
LIN {X 0,Y 551.82,Z 763.241,A -85,B 0,C 180,E1 -3425.481,E2 -3425.481} C_VEL
LIN {X 0,Y 551.921,Z 756.919,A -85,B 0,C 180,E1 -3426.431,E2 -3426.431} C_VEL
LIN {X 0,Y 551.997,Z 749.525,A -85,B 0,C 180,E1 -3427.315,E2 -3427.315} C_VEL
LIN {X 0,Y 552.121,Z 740.87,A -85,B 0,C 180,E1 -3428.141,E2 -3428.141} C_VEL
LIN {X 0,Y 552.323,Z 730.99,A -85,B 0,C 180,E1 -3428.875,E2 -3428.875} C_VEL
LIN {X 0,Y 552.406,Z 721.415,A -85,B 0,C 180,E1 -3429.428,E2 -3429.428} C_VEL
LIN {X 0,Y 552.526,Z 710.785,A -85,B 0,C 180,E1 -3429.888,E2 -3429.888} C_VEL
LIN {X 0,Y 552.581,Z 699.097,A -85,B 0,C 180,E1 -3430.234,E2 -3430.234} C_VEL
LIN {X 0,Y 552.688,Z 684.585,A -85,B 0,C 180,E1 -3430.463,E2 -3430.463} C_VEL
LIN {X 0,Y 552.647,Z 620.389,A -85,B 0,C 180,E1 -3431.296,E2 -3431.296} C_VEL
LIN {X 0,Y 552.166,Z 616.244,A -85,B 0,C 180,E1 -3431.39,E2 -3431.39} C_VEL
LIN {X 0,Y 552.435,Z 594.305,A -85,B 0,C 180,E1 -3434.364,E2 -3434.364} C_VEL
LIN {X 0,Y 552.737,Z 571.458,A -85,B 0,C 180,E1 -3437.518,E2 -3437.518} C_VEL
LIN {X 0,Y 552.992,Z 557.228,A -85,B 0,C 180,E1 -3439.506,E2 -3439.506} C_VEL
LIN {X 0,Y 552.443,Z 553.841,A -85,B 0,C 180,E1 -3440.002,E2 -3440.002} C_VEL
LIN {X 0,Y 549.654,Z 548.515,A -85,B 0,C 180,E1 -3440.825,E2 -3440.825} C_VEL
LIN {X 0,Y 546.851,Z 543.213,A -85,B 0,C 180,E1 -3441.657,E2 -3441.657} C_VEL
LIN {X 0,Y 546.289,Z 539.773,A -85,B 0,C 180,E1 -3442.16,E2 -3442.16} C_VEL
LIN {X 0,Y 546.52,Z 524.464,A -85,B 0,C 180,E1 -3444.3,E2 -3444.3} C_VEL
LIN {X 0,Y 545.13,Z 516.705,A -85,B 0,C 180,E1 -3445.473,E2 -3445.473} C_VEL
LIN {X 0,Y 545.106,Z 516.582,A -85,B 0,C 180,E1 -3448.492,E2 -3448.492} C_VEL
LIN {X 0,Y 545.069,Z 516.586,A -85,B 0,C 180,E1 -3451.048,E2 -3451.048} C_VEL
LIN {X 0,Y 545.071,Z 516.593,A -85,B 0,C 180,E1 -3453.672,E2 -3453.672} C_VEL
LIN {X 0,Y 545.076,Z 516.584,A -85,B 0,C 180,E1 -3456.926,E2 -3456.926} C_VEL
LIN {X 0,Y 545.071,Z 516.58,A -85,B 0,C 180,E1 -3460.142,E2 -3460.142} C_VEL
LIN {X 0,Y 545.066,Z 516.574,A -85,B 0,C 180,E1 -3462.697,E2 -3462.697} C_VEL
LIN {X 0,Y 545.062,Z 516.587,A -85,B 0,C 180,E1 -3465.871,E2 -3465.871} C_VEL
LIN {X 0,Y 545.087,Z 516.584,A -85,B 0,C 180,E1 -3468.885,E2 -3468.885} C_VEL
LIN {X 0,Y 545.054,Z 516.586,A -85,B 0,C 180,E1 -3471.864,E2 -3471.864} C_VEL
LIN {X 0,Y 545.041,Z 516.589,A -85,B 0,C 180,E1 -3474.531,E2 -3474.531} C_VEL
LIN {X 0,Y 545.07,Z 516.591,A -85,B 0,C 180,E1 -3477.211,E2 -3477.211} C_VEL
LIN {X 0,Y 545.069,Z 516.585,A -85,B 0,C 180,E1 -3479.81,E2 -3479.81} C_VEL
LIN {X 0,Y 545.086,Z 516.584,A -85,B 0,C 180,E1 -3482.344,E2 -3482.344} C_VEL
LIN {X 0,Y 545.122,Z 516.585,A -85,B 0,C 180,E1 -3484.82,E2 -3484.82} C_VEL
LIN {X 0,Y 545.041,Z 516.591,A -85,B 0,C 180,E1 -3487.242,E2 -3487.242} C_VEL
LIN {X 0,Y 545.153,Z 516.755,A -85,B 0,C 180,E1 -3489.827,E2 -3489.827} C_VEL
LIN {X 0,Y 545.626,Z 521.841,A -85,B 0,C 180,E1 -3490.824,E2 -3490.824} C_VEL
LIN {X 0,Y 545.367,Z 536.386,A -85,B 0,C 180,E1 -3493.53,E2 -3493.53} C_VEL
LIN {X 0,Y 545.179,Z 546.321,A -85,B 0,C 180,E1 -3495.326,E2 -3495.326} C_VEL
LIN {X 0,Y 545.289,Z 548.012,A -85,B 0,C 180,E1 -3495.504,E2 -3495.504} C_VEL
LIN {X 0,Y 546.565,Z 555.59,A -85,B 0,C 180,E1 -3495.649,E2 -3495.649} C_VEL
LIN {X 0,Y 546.232,Z 654.031,A -85,B 0,C 180,E1 -3496.963,E2 -3496.963} C_VEL
LIN {X 0,Y 546.076,Z 667.276,A -85,B 0,C 180,E1 -3497.291,E2 -3497.291} C_VEL
LIN {X 0,Y 545.899,Z 679.415,A -85,B 0,C 180,E1 -3497.735,E2 -3497.735} C_VEL
LIN {X 0,Y 545.728,Z 691.608,A -85,B 0,C 180,E1 -3498.342,E2 -3498.342} C_VEL
LIN {X 0,Y 545.534,Z 702.571,A -85,B 0,C 180,E1 -3499.045,E2 -3499.045} C_VEL
LIN {X 0,Y 545.266,Z 713.087,A -85,B 0,C 180,E1 -3499.885,E2 -3499.885} C_VEL
LIN {X 0,Y 545.122,Z 721.683,A -85,B 0,C 180,E1 -3500.725,E2 -3500.725} C_VEL
LIN {X 0,Y 544.976,Z 729.601,A -85,B 0,C 180,E1 -3501.658,E2 -3501.658} C_VEL
LIN {X 0,Y 544.828,Z 737.347,A -85,B 0,C 180,E1 -3502.774,E2 -3502.774} C_VEL
LIN {X 0,Y 544.778,Z 744.458,A -85,B 0,C 180,E1 -3504.076,E2 -3504.076} C_VEL
LIN {X 0,Y 544.629,Z 749.199,A -85,B 0,C 180,E1 -3505.188,E2 -3505.188} C_VEL
LIN {X 0,Y 544.669,Z 752.83,A -85,B 0,C 180,E1 -3506.3,E2 -3506.3} C_VEL
LIN {X 0,Y 544.65,Z 754.707,A -85,B 0,C 180,E1 -3507.041,E2 -3507.041} C_VEL
LIN {X 0,Y 544.571,Z 756.129,A -85,B 0,C 180,E1 -3507.781,E2 -3507.781} C_VEL
LIN {X 0,Y 544.542,Z 757.757,A -85,B 0,C 180,E1 -3509.26,E2 -3509.26} C_VEL
LIN {X 0,Y 544.542,Z 757.996,A -85,B 0,C 180,E1 -3509.999,E2 -3509.999} C_VEL
LIN {X 0,Y 544.542,Z 757.815,A -85,B 0,C 180,E1 -3510.739,E2 -3510.739} C_VEL
LIN {X 0,Y 544.571,Z 756.267,A -85,B 0,C 180,E1 -3512.218,E2 -3512.218} C_VEL
LIN {X 0,Y 544.651,Z 754.906,A -85,B 0,C 180,E1 -3512.958,E2 -3512.958} C_VEL
LIN {X 0,Y 544.684,Z 752.026,A -85,B 0,C 180,E1 -3514.069,E2 -3514.069} C_VEL
LIN {X 0,Y 544.653,Z 748.125,A -85,B 0,C 180,E1 -3515.182,E2 -3515.182} C_VEL
LIN {X 0,Y 544.724,Z 742.9,A -85,B 0,C 180,E1 -3516.335,E2 -3516.335} C_VEL
LIN {X 0,Y 544.858,Z 735.537,A -85,B 0,C 180,E1 -3517.597,E2 -3517.597} C_VEL
LIN {X 0,Y 545.025,Z 727.353,A -85,B 0,C 180,E1 -3518.714,E2 -3518.714} C_VEL
LIN {X 0,Y 545.157,Z 718.985,A -85,B 0,C 180,E1 -3519.647,E2 -3519.647} C_VEL
LIN {X 0,Y 545.389,Z 708.667,A -85,B 0,C 180,E1 -3520.58,E2 -3520.58} C_VEL
LIN {X 0,Y 545.647,Z 697.333,A -85,B 0,C 180,E1 -3521.4,E2 -3521.4} C_VEL
LIN {X 0,Y 545.787,Z 687.261,A -85,B 0,C 180,E1 -3521.983,E2 -3521.983} C_VEL
LIN {X 0,Y 545.981,Z 674.738,A -85,B 0,C 180,E1 -3522.545,E2 -3522.545} C_VEL
LIN {X 0,Y 546.139,Z 661.297,A -85,B 0,C 180,E1 -3522.967,E2 -3522.967} C_VEL
LIN {X 0,Y 546.288,Z 647.974,A -85,B 0,C 180,E1 -3523.223,E2 -3523.223} C_VEL
LIN {X 0,Y 546.433,Z 554.456,A -85,B 0,C 180,E1 -3524.459,E2 -3524.459} C_VEL
LIN {X 0,Y 545.259,Z 547.716,A -85,B 0,C 180,E1 -3524.6,E2 -3524.6} C_VEL
LIN {X 0,Y 545.229,Z 545.273,A -85,B 0,C 180,E1 -3524.939,E2 -3524.939} C_VEL
LIN {X 0,Y 545.533,Z 528.563,A -85,B 0,C 180,E1 -3528.009,E2 -3528.009} C_VEL
LIN {X 0,Y 545.465,Z 518.774,A -85,B 0,C 180,E1 -3529.853,E2 -3529.853} C_VEL
LIN {X 0,Y 545.124,Z 516.676,A -85,B 0,C 180,E1 -3530.293,E2 -3530.293} C_VEL
LIN {X 0,Y 545.093,Z 516.587,A -85,B 0,C 180,E1 -3533.558,E2 -3533.558} C_VEL
LIN {X 0,Y 545.08,Z 516.583,A -85,B 0,C 180,E1 -3536,E2 -3536} C_VEL
LIN {X 0,Y 545.089,Z 516.582,A -85,B 0,C 180,E1 -3538.747,E2 -3538.747} C_VEL
LIN {X 0,Y 545.077,Z 516.588,A -85,B 0,C 180,E1 -3541.682,E2 -3541.682} C_VEL
LIN {X 0,Y 545.08,Z 516.583,A -85,B 0,C 180,E1 -3544.562,E2 -3544.562} C_VEL
LIN {X 0,Y 545.039,Z 516.594,A -85,B 0,C 180,E1 -3547.303,E2 -3547.303} C_VEL
LIN {X 0,Y 545.072,Z 516.582,A -85,B 0,C 180,E1 -3550.141,E2 -3550.141} C_VEL
LIN {X 0,Y 545.084,Z 516.586,A -85,B 0,C 180,E1 -3553.105,E2 -3553.105} C_VEL
LIN {X 0,Y 545.063,Z 516.584,A -85,B 0,C 180,E1 -3556.223,E2 -3556.223} C_VEL
LIN {X 0,Y 545.097,Z 516.582,A -85,B 0,C 180,E1 -3558.887,E2 -3558.887} C_VEL
LIN {X 0,Y 545.05,Z 516.587,A -85,B 0,C 180,E1 -3561.762,E2 -3561.762} C_VEL
LIN {X 0,Y 545.061,Z 516.584,A -85,B 0,C 180,E1 -3564.533,E2 -3564.533} C_VEL
LIN {X 0,Y 545.078,Z 516.588,A -85,B 0,C 180,E1 -3567.212,E2 -3567.212} C_VEL
LIN {X 0,Y 545.096,Z 516.584,A -85,B 0,C 180,E1 -3569.812,E2 -3569.812} C_VEL
LIN {X 0,Y 545.096,Z 516.579,A -85,B 0,C 180,E1 -3572.824,E2 -3572.824} C_VEL
LIN {X 0,Y 545.047,Z 516.593,A -85,B 0,C 180,E1 -3575.63,E2 -3575.63} C_VEL
LIN {X 0,Y 545.063,Z 516.583,A -85,B 0,C 180,E1 -3578.836,E2 -3578.836} C_VEL
LIN {X 0,Y 545.079,Z 516.587,A -85,B 0,C 180,E1 -3581.195,E2 -3581.195} C_VEL
LIN {X 0,Y 545.071,Z 516.589,A -85,B 0,C 180,E1 -3583.521,E2 -3583.521} C_VEL
LIN {X 0,Y 545.088,Z 516.586,A -85,B 0,C 180,E1 -3585.82,E2 -3585.82} C_VEL
LIN {X 0,Y 545.111,Z 516.578,A -85,B 0,C 180,E1 -3588.849,E2 -3588.849} C_VEL
LIN {X 0,Y 545.127,Z 516.581,A -85,B 0,C 180,E1 -3591.847,E2 -3591.847} C_VEL
LIN {X 0,Y 545.201,Z 516.567,A -85,B 0,C 180,E1 -3594.823,E2 -3594.823} C_VEL
LIN {X 0,Y 545.189,Z 516.573,A -85,B 0,C 180,E1 -3597.784,E2 -3597.784} C_VEL
LIN {X 0,Y 545.209,Z 516.566,A -85,B 0,C 180,E1 -3600.739,E2 -3600.739} C_VEL
LIN {X 0,Y 545.17,Z 516.571,A -85,B 0,C 180,E1 -3602.956,E2 -3602.956} C_VEL
LIN {X 0,Y 545.164,Z 516.576,A -85,B 0,C 180,E1 -3605.92,E2 -3605.92} C_VEL
LIN {X 0,Y 545.115,Z 516.578,A -85,B 0,C 180,E1 -3608.9,E2 -3608.9} C_VEL
LIN {X 0,Y 545.128,Z 516.581,A -85,B 0,C 180,E1 -3611.904,E2 -3611.904} C_VEL
LIN {X 0,Y 545.078,Z 516.583,A -85,B 0,C 180,E1 -3614.944,E2 -3614.944} C_VEL
LIN {X 0,Y 545.076,Z 516.586,A -85,B 0,C 180,E1 -3618.026,E2 -3618.026} C_VEL
LIN {X 0,Y 545.092,Z 516.58,A -85,B 0,C 180,E1 -3620.372,E2 -3620.372} C_VEL
LIN {X 0,Y 545.085,Z 516.589,A -85,B 0,C 180,E1 -3623.559,E2 -3623.559} C_VEL
LIN {X 0,Y 545.082,Z 516.584,A -85,B 0,C 180,E1 -3626,E2 -3626} C_VEL
LIN {X 0,Y 545.084,Z 516.582,A -85,B 0,C 180,E1 -3628.749,E2 -3628.749} C_VEL
LIN {X 0,Y 545.073,Z 516.592,A -85,B 0,C 180,E1 -3631.683,E2 -3631.683} C_VEL
LIN {X 0,Y 545.08,Z 516.581,A -85,B 0,C 180,E1 -3634.563,E2 -3634.563} C_VEL
LIN {X 0,Y 545.034,Z 516.587,A -85,B 0,C 180,E1 -3637.304,E2 -3637.304} C_VEL
LIN {X 0,Y 545.07,Z 516.586,A -85,B 0,C 180,E1 -3640.142,E2 -3640.142} C_VEL
LIN {X 0,Y 545.074,Z 516.581,A -85,B 0,C 180,E1 -3643.107,E2 -3643.107} C_VEL
LIN {X 0,Y 545.063,Z 516.585,A -85,B 0,C 180,E1 -3646.225,E2 -3646.225} C_VEL
LIN {X 0,Y 545.098,Z 516.581,A -85,B 0,C 180,E1 -3648.888,E2 -3648.888} C_VEL
LIN {X 0,Y 545.052,Z 516.587,A -85,B 0,C 180,E1 -3651.764,E2 -3651.764} C_VEL
LIN {X 0,Y 545.051,Z 516.587,A -85,B 0,C 180,E1 -3654.534,E2 -3654.534} C_VEL
LIN {X 0,Y 545.08,Z 516.581,A -85,B 0,C 180,E1 -3657.213,E2 -3657.213} C_VEL
LIN {X 0,Y 545.065,Z 516.577,A -85,B 0,C 180,E1 -3659.812,E2 -3659.812} C_VEL
LIN {X 0,Y 545.091,Z 516.581,A -85,B 0,C 180,E1 -3662.345,E2 -3662.345} C_VEL
LIN {X 0,Y 545.117,Z 516.579,A -85,B 0,C 180,E1 -3664.821,E2 -3664.821} C_VEL
LIN {X 0,Y 545.131,Z 516.812,A -85,B 0,C 180,E1 -3666.308,E2 -3666.308} C_VEL
LIN {X 0,Y 546.295,Z 523.853,A -85,B 0,C 180,E1 -3667.472,E2 -3667.472} C_VEL
LIN {X 0,Y 545.9,Z 543.109,A -85,B 0,C 180,E1 -3670.445,E2 -3670.445} C_VEL
LIN {X 0,Y 545.579,Z 560.843,A -85,B 0,C 180,E1 -3673.152,E2 -3673.152} C_VEL
LIN {X 0,Y 545.405,Z 575.941,A -85,B 0,C 180,E1 -3675.417,E2 -3675.417} C_VEL
LIN {X 0,Y 546.332,Z 582.179,A -85,B 0,C 180,E1 -3675.553,E2 -3675.553} C_VEL
LIN {X 0,Y 546.54,Z 592.434,A -85,B 0,C 180,E1 -3675.695,E2 -3675.695} C_VEL
LIN {X 0,Y 546.239,Z 683.981,A -85,B 0,C 180,E1 -3676.918,E2 -3676.918} C_VEL
LIN {X 0,Y 546.076,Z 697.233,A -85,B 0,C 180,E1 -3677.245,E2 -3677.245} C_VEL
LIN {X 0,Y 545.898,Z 710.498,A -85,B 0,C 180,E1 -3677.736,E2 -3677.736} C_VEL
LIN {X 0,Y 545.726,Z 722.379,A -85,B 0,C 180,E1 -3678.342,E2 -3678.342} C_VEL
LIN {X 0,Y 545.521,Z 733.207,A -85,B 0,C 180,E1 -3679.046,E2 -3679.046} C_VEL
LIN {X 0,Y 545.258,Z 743.612,A -85,B 0,C 180,E1 -3679.886,E2 -3679.886} C_VEL
LIN {X 0,Y 545.084,Z 752.12,A -85,B 0,C 180,E1 -3680.726,E2 -3680.726} C_VEL
LIN {X 0,Y 544.977,Z 759.966,A -85,B 0,C 180,E1 -3681.659,E2 -3681.659} C_VEL
LIN {X 0,Y 544.823,Z 767.626,A -85,B 0,C 180,E1 -3682.775,E2 -3682.775} C_VEL
LIN {X 0,Y 544.776,Z 774.682,A -85,B 0,C 180,E1 -3684.077,E2 -3684.077} C_VEL
LIN {X 0,Y 544.629,Z 779.374,A -85,B 0,C 180,E1 -3685.189,E2 -3685.189} C_VEL
LIN {X 0,Y 544.669,Z 782.962,A -85,B 0,C 180,E1 -3686.302,E2 -3686.302} C_VEL
LIN {X 0,Y 544.65,Z 784.811,A -85,B 0,C 180,E1 -3687.042,E2 -3687.042} C_VEL
LIN {X 0,Y 544.546,Z 787.185,A -85,B 0,C 180,E1 -3688.522,E2 -3688.522} C_VEL
LIN {X 0,Y 544.541,Z 788,A -85,B 0,C 180,E1 -3690.001,E2 -3690.001} C_VEL
LIN {X 0,Y 544.546,Z 787.183,A -85,B 0,C 180,E1 -3691.48,E2 -3691.48} C_VEL
LIN {X 0,Y 544.651,Z 784.806,A -85,B 0,C 180,E1 -3692.959,E2 -3692.959} C_VEL
LIN {X 0,Y 544.684,Z 781.893,A -85,B 0,C 180,E1 -3694.07,E2 -3694.07} C_VEL
LIN {X 0,Y 544.654,Z 777.947,A -85,B 0,C 180,E1 -3695.183,E2 -3695.183} C_VEL
LIN {X 0,Y 544.74,Z 772.703,A -85,B 0,C 180,E1 -3696.328,E2 -3696.328} C_VEL
LIN {X 0,Y 544.837,Z 766.463,A -85,B 0,C 180,E1 -3697.412,E2 -3697.412} C_VEL
LIN {X 0,Y 545.007,Z 758.473,A -85,B 0,C 180,E1 -3698.529,E2 -3698.529} C_VEL
LIN {X 0,Y 545.153,Z 750.328,A -85,B 0,C 180,E1 -3699.461,E2 -3699.461} C_VEL
LIN {X 0,Y 545.34,Z 740.393,A -85,B 0,C 180,E1 -3700.395,E2 -3700.395} C_VEL
LIN {X 0,Y 545.567,Z 729.584,A -85,B 0,C 180,E1 -3701.208,E2 -3701.208} C_VEL
LIN {X 0,Y 545.743,Z 718.162,A -85,B 0,C 180,E1 -3701.891,E2 -3701.891} C_VEL
LIN {X 0,Y 545.95,Z 705.969,A -85,B 0,C 180,E1 -3702.453,E2 -3702.453} C_VEL
LIN {X 0,Y 546.137,Z 693.161,A -85,B 0,C 180,E1 -3702.873,E2 -3702.873} C_VEL
LIN {X 0,Y 546.256,Z 679.566,A -85,B 0,C 180,E1 -3703.154,E2 -3703.154} C_VEL
LIN {X 0,Y 546.438,Z 582.886,A -85,B 0,C 180,E1 -3704.435,E2 -3704.435} C_VEL
LIN {X 0,Y 545.416,Z 575.984,A -85,B 0,C 180,E1 -3704.58,E2 -3704.58} C_VEL
LIN {X 0,Y 545.681,Z 555.771,A -85,B 0,C 180,E1 -3707.622,E2 -3707.622} C_VEL
LIN {X 0,Y 546.062,Z 535.458,A -85,B 0,C 180,E1 -3710.729,E2 -3710.729} C_VEL
LIN {X 0,Y 546.239,Z 522.716,A -85,B 0,C 180,E1 -3712.705,E2 -3712.705} C_VEL
LIN {X 0,Y 545.1,Z 516.711,A -85,B 0,C 180,E1 -3713.736,E2 -3713.736} C_VEL
LIN {X 0,Y 545.083,Z 516.583,A -85,B 0,C 180,E1 -3716.001,E2 -3716.001} C_VEL
LIN {X 0,Y 545.093,Z 516.579,A -85,B 0,C 180,E1 -3718.748,E2 -3718.748} C_VEL
LIN {X 0,Y 545.062,Z 516.587,A -85,B 0,C 180,E1 -3721.679,E2 -3721.679} C_VEL
LIN {X 0,Y 545.066,Z 516.589,A -85,B 0,C 180,E1 -3724.565,E2 -3724.565} C_VEL
LIN {X 0,Y 545.04,Z 516.588,A -85,B 0,C 180,E1 -3727.304,E2 -3727.304} C_VEL
LIN {X 0,Y 545.069,Z 516.593,A -85,B 0,C 180,E1 -3730.143,E2 -3730.143} C_VEL
LIN {X 0,Y 545.082,Z 516.583,A -85,B 0,C 180,E1 -3733.107,E2 -3733.107} C_VEL
LIN {X 0,Y 545.053,Z 516.594,A -85,B 0,C 180,E1 -3736.226,E2 -3736.226} C_VEL
LIN {X 0,Y 545.084,Z 516.583,A -85,B 0,C 180,E1 -3738.885,E2 -3738.885} C_VEL
LIN {X 0,Y 545.085,Z 516.584,A -85,B 0,C 180,E1 -3740.819,E2 -3740.819} C_VEL
LIN {X 0,Y 545.053,Z 516.589,A -85,B 0,C 180,E1 -3743.62,E2 -3743.62} C_VEL
LIN {X 0,Y 545.071,Z 516.592,A -85,B 0,C 180,E1 -3746.328,E2 -3746.328} C_VEL
LIN {X 0,Y 545.069,Z 516.586,A -85,B 0,C 180,E1 -3748.952,E2 -3748.952} C_VEL
LIN {X 0,Y 545.106,Z 516.582,A -85,B 0,C 180,E1 -3751.508,E2 -3751.508} C_VEL
LIN {X 0,Y 545.099,Z 516.589,A -85,B 0,C 180,E1 -3754.491,E2 -3754.491} C_VEL
LIN {X 0,Y 545.165,Z 516.844,A -85,B 0,C 180,E1 -3754.874,E2 -3754.874} C_VEL
LIN {X 0,Y 546.423,Z 524.548,A -85,B 0,C 180,E1 -3755.95,E2 -3755.95} C_VEL
LIN {X 0,Y 546.227,Z 542.009,A -85,B 0,C 180,E1 -3758.29,E2 -3758.29} C_VEL
LIN {X 0,Y 545.962,Z 560.516,A -85,B 0,C 180,E1 -3760.837,E2 -3760.837} C_VEL
LIN {X 0,Y 545.659,Z 578.607,A -85,B 0,C 180,E1 -3763.347,E2 -3763.347} C_VEL
LIN {X 0,Y 545.352,Z 599.127,A -85,B 0,C 180,E1 -3766.207,E2 -3766.207} C_VEL
LIN {X 0,Y 545.122,Z 616.427,A -85,B 0,C 180,E1 -3768.563,E2 -3768.563} C_VEL
LIN {X 0,Y 545.811,Z 622.919,A -85,B 0,C 180,E1 -3768.685,E2 -3768.685} C_VEL
LIN {X 0,Y 545.686,Z 695.821,A -85,B 0,C 180,E1 -3769.659,E2 -3769.659} C_VEL
LIN {X 0,Y 545.545,Z 706.81,A -85,B 0,C 180,E1 -3769.938,E2 -3769.938} C_VEL
LIN {X 0,Y 545.418,Z 717.63,A -85,B 0,C 180,E1 -3770.357,E2 -3770.357} C_VEL
LIN {X 0,Y 545.269,Z 728.08,A -85,B 0,C 180,E1 -3770.915,E2 -3770.915} C_VEL
LIN {X 0,Y 545.132,Z 737.475,A -85,B 0,C 180,E1 -3771.567,E2 -3771.567} C_VEL
LIN {X 0,Y 544.97,Z 746.882,A -85,B 0,C 180,E1 -3772.404,E2 -3772.404} C_VEL
LIN {X 0,Y 544.881,Z 755.057,A -85,B 0,C 180,E1 -3773.334,E2 -3773.334} C_VEL
LIN {X 0,Y 544.817,Z 761.548,A -85,B 0,C 180,E1 -3774.262,E2 -3774.262} C_VEL
LIN {X 0,Y 544.704,Z 766.726,A -85,B 0,C 180,E1 -3775.189,E2 -3775.189} C_VEL
LIN {X 0,Y 544.677,Z 771.461,A -85,B 0,C 180,E1 -3776.301,E2 -3776.301} C_VEL
LIN {X 0,Y 544.661,Z 773.824,A -85,B 0,C 180,E1 -3777.041,E2 -3777.041} C_VEL
LIN {X 0,Y 544.571,Z 775.618,A -85,B 0,C 180,E1 -3777.781,E2 -3777.781} C_VEL
LIN {X 0,Y 544.543,Z 776.913,A -85,B 0,C 180,E1 -3778.521,E2 -3778.521} C_VEL
LIN {X 0,Y 544.538,Z 777.709,A -85,B 0,C 180,E1 -3779.261,E2 -3779.261} C_VEL
LIN {X 0,Y 544.539,Z 777.996,A -85,B 0,C 180,E1 -3780,E2 -3780} C_VEL
LIN {X 0,Y 544.54,Z 777.775,A -85,B 0,C 180,E1 -3780.74,E2 -3780.74} C_VEL
LIN {X 0,Y 544.547,Z 777.042,A -85,B 0,C 180,E1 -3781.479,E2 -3781.479} C_VEL
LIN {X 0,Y 544.572,Z 775.803,A -85,B 0,C 180,E1 -3782.219,E2 -3782.219} C_VEL
LIN {X 0,Y 544.691,Z 772.983,A -85,B 0,C 180,E1 -3783.329,E2 -3783.329} C_VEL
LIN {X 0,Y 544.706,Z 768.864,A -85,B 0,C 180,E1 -3784.44,E2 -3784.44} C_VEL
LIN {X 0,Y 544.763,Z 763.238,A -85,B 0,C 180,E1 -3785.553,E2 -3785.553} C_VEL
LIN {X 0,Y 544.847,Z 756.553,A -85,B 0,C 180,E1 -3786.562,E2 -3786.562} C_VEL
LIN {X 0,Y 544.932,Z 749.527,A -85,B 0,C 180,E1 -3787.41,E2 -3787.41} C_VEL
LIN {X 0,Y 545.082,Z 740.864,A -85,B 0,C 180,E1 -3788.247,E2 -3788.247} C_VEL
LIN {X 0,Y 545.307,Z 730.988,A -85,B 0,C 180,E1 -3788.99,E2 -3788.99} C_VEL
LIN {X 0,Y 545.413,Z 721.418,A -85,B 0,C 180,E1 -3789.55,E2 -3789.55} C_VEL
LIN {X 0,Y 545.545,Z 710.786,A -85,B 0,C 180,E1 -3790.016,E2 -3790.016} C_VEL
LIN {X 0,Y 545.602,Z 699.066,A -85,B 0,C 180,E1 -3790.366,E2 -3790.366} C_VEL
LIN {X 0,Y 545.722,Z 684.539,A -85,B 0,C 180,E1 -3790.598,E2 -3790.598} C_VEL
LIN {X 0,Y 545.661,Z 620.939,A -85,B 0,C 180,E1 -3791.435,E2 -3791.435} C_VEL
LIN {X 0,Y 545.141,Z 616.285,A -85,B 0,C 180,E1 -3791.536,E2 -3791.536} C_VEL
LIN {X 0,Y 545.439,Z 594.569,A -85,B 0,C 180,E1 -3794.515,E2 -3794.515} C_VEL
LIN {X 0,Y 545.801,Z 571.363,A -85,B 0,C 180,E1 -3797.761,E2 -3797.761} C_VEL
LIN {X 0,Y 546.154,Z 550.009,A -85,B 0,C 180,E1 -3800.725,E2 -3800.725} C_VEL
LIN {X 0,Y 546.289,Z 539.773,A -85,B 0,C 180,E1 -3802.16,E2 -3802.16} C_VEL
LIN {X 0,Y 545.797,Z 536.35,A -85,B 0,C 180,E1 -3802.661,E2 -3802.661} C_VEL
LIN {X 0,Y 543.195,Z 531.061,A -85,B 0,C 180,E1 -3803.498,E2 -3803.498} C_VEL
LIN {X 0,Y 539.715,Z 524.744,A -85,B 0,C 180,E1 -3804.516,E2 -3804.516} C_VEL
LIN {X 0,Y 539.061,Z 522.492,A -85,B 0,C 180,E1 -3804.86,E2 -3804.86} C_VEL
LIN {X 0,Y 538.066,Z 517.557,A -85,B 0,C 180,E1 -3805.642,E2 -3805.642} C_VEL
LIN {X 0,Y 538.048,Z 517.466,A -85,B 0,C 180,E1 -3808.05,E2 -3808.05} C_VEL
LIN {X 0,Y 538.024,Z 517.463,A -85,B 0,C 180,E1 -3810.627,E2 -3810.627} C_VEL
LIN {X 0,Y 538.049,Z 517.463,A -85,B 0,C 180,E1 -3813.283,E2 -3813.283} C_VEL
LIN {X 0,Y 538.004,Z 517.468,A -85,B 0,C 180,E1 -3816.004,E2 -3816.004} C_VEL
LIN {X 0,Y 538.018,Z 517.463,A -85,B 0,C 180,E1 -3818.83,E2 -3818.83} C_VEL
LIN {X 0,Y 538.034,Z 517.453,A -85,B 0,C 180,E1 -3821.773,E2 -3821.773} C_VEL
LIN {X 0,Y 538.011,Z 517.462,A -85,B 0,C 180,E1 -3824.862,E2 -3824.862} C_VEL
LIN {X 0,Y 538.024,Z 517.47,A -85,B 0,C 180,E1 -3827.214,E2 -3827.214} C_VEL
LIN {X 0,Y 538.015,Z 517.454,A -85,B 0,C 180,E1 -3830.202,E2 -3830.202} C_VEL
LIN {X 0,Y 538.029,Z 517.468,A -85,B 0,C 180,E1 -3833.067,E2 -3833.067} C_VEL
LIN {X 0,Y 538.015,Z 517.462,A -85,B 0,C 180,E1 -3835.826,E2 -3835.826} C_VEL
LIN {X 0,Y 538.013,Z 517.465,A -85,B 0,C 180,E1 -3838.498,E2 -3838.498} C_VEL
LIN {X 0,Y 538.065,Z 517.463,A -85,B 0,C 180,E1 -3841.1,E2 -3841.1} C_VEL
LIN {X 0,Y 538.046,Z 517.461,A -85,B 0,C 180,E1 -3843.633,E2 -3843.633} C_VEL
LIN {X 0,Y 538.012,Z 517.462,A -85,B 0,C 180,E1 -3846.122,E2 -3846.122} C_VEL
LIN {X 0,Y 538.057,Z 517.464,A -85,B 0,C 180,E1 -3849.349,E2 -3849.349} C_VEL
LIN {X 0,Y 538.116,Z 517.638,A -85,B 0,C 180,E1 -3849.693,E2 -3849.693} C_VEL
LIN {X 0,Y 538.671,Z 523.032,A -85,B 0,C 180,E1 -3850.765,E2 -3850.765} C_VEL
LIN {X 0,Y 538.349,Z 538.597,A -85,B 0,C 180,E1 -3853.699,E2 -3853.699} C_VEL
LIN {X 0,Y 538.25,Z 544.993,A -85,B 0,C 180,E1 -3854.862,E2 -3854.862} C_VEL
LIN {X 0,Y 538.303,Z 548.254,A -85,B 0,C 180,E1 -3855.301,E2 -3855.301} C_VEL
LIN {X 0,Y 539.681,Z 556.842,A -85,B 0,C 180,E1 -3855.478,E2 -3855.478} C_VEL
LIN {X 0,Y 539.328,Z 654.06,A -85,B 0,C 180,E1 -3856.794,E2 -3856.794} C_VEL
LIN {X 0,Y 539.164,Z 667.295,A -85,B 0,C 180,E1 -3857.125,E2 -3857.125} C_VEL
LIN {X 0,Y 538.951,Z 679.428,A -85,B 0,C 180,E1 -3857.574,E2 -3857.574} C_VEL
LIN {X 0,Y 538.746,Z 691.616,A -85,B 0,C 180,E1 -3858.188,E2 -3858.188} C_VEL
LIN {X 0,Y 538.542,Z 702.578,A -85,B 0,C 180,E1 -3858.901,E2 -3858.901} C_VEL
LIN {X 0,Y 538.278,Z 713.093,A -85,B 0,C 180,E1 -3859.752,E2 -3859.752} C_VEL
LIN {X 0,Y 538.086,Z 721.688,A -85,B 0,C 180,E1 -3860.603,E2 -3860.603} C_VEL
LIN {X 0,Y 537.923,Z 729.606,A -85,B 0,C 180,E1 -3861.547,E2 -3861.547} C_VEL
LIN {X 0,Y 537.759,Z 737.351,A -85,B 0,C 180,E1 -3862.679,E2 -3862.679} C_VEL
LIN {X 0,Y 537.694,Z 744.461,A -85,B 0,C 180,E1 -3863.997,E2 -3863.997} C_VEL
LIN {X 0,Y 537.54,Z 749.201,A -85,B 0,C 180,E1 -3865.124,E2 -3865.124} C_VEL
LIN {X 0,Y 537.591,Z 752.831,A -85,B 0,C 180,E1 -3866.252,E2 -3866.252} C_VEL
LIN {X 0,Y 537.551,Z 754.709,A -85,B 0,C 180,E1 -3867.002,E2 -3867.002} C_VEL
LIN {X 0,Y 537.49,Z 756.129,A -85,B 0,C 180,E1 -3867.751,E2 -3867.751} C_VEL
LIN {X 0,Y 537.442,Z 757.757,A -85,B 0,C 180,E1 -3869.25,E2 -3869.25} C_VEL
LIN {X 0,Y 537.442,Z 757.996,A -85,B 0,C 180,E1 -3869.999,E2 -3869.999} C_VEL
LIN {X 0,Y 537.442,Z 757.814,A -85,B 0,C 180,E1 -3870.749,E2 -3870.749} C_VEL
LIN {X 0,Y 537.49,Z 756.266,A -85,B 0,C 180,E1 -3872.247,E2 -3872.247} C_VEL
LIN {X 0,Y 537.552,Z 754.904,A -85,B 0,C 180,E1 -3872.997,E2 -3872.997} C_VEL
LIN {X 0,Y 537.604,Z 752.023,A -85,B 0,C 180,E1 -3874.122,E2 -3874.122} C_VEL
LIN {X 0,Y 537.587,Z 748.122,A -85,B 0,C 180,E1 -3875.25,E2 -3875.25} C_VEL
LIN {X 0,Y 537.638,Z 743.37,A -85,B 0,C 180,E1 -3876.32,E2 -3876.32} C_VEL
LIN {X 0,Y 537.789,Z 736.762,A -85,B 0,C 180,E1 -3877.508,E2 -3877.508} C_VEL
LIN {X 0,Y 537.969,Z 728.836,A -85,B 0,C 180,E1 -3878.64,E2 -3878.64} C_VEL
LIN {X 0,Y 538.112,Z 720.763,A -85,B 0,C 180,E1 -3879.585,E2 -3879.585} C_VEL
LIN {X 0,Y 538.347,Z 710.91,A -85,B 0,C 180,E1 -3880.53,E2 -3880.53} C_VEL
LIN {X 0,Y 538.58,Z 701.23,A -85,B 0,C 180,E1 -3881.287,E2 -3881.287} C_VEL
LIN {X 0,Y 538.742,Z 690.722,A -85,B 0,C 180,E1 -3881.954,E2 -3881.954} C_VEL
LIN {X 0,Y 538.988,Z 678.192,A -85,B 0,C 180,E1 -3882.567,E2 -3882.567} C_VEL
LIN {X 0,Y 539.181,Z 664.86,A -85,B 0,C 180,E1 -3883.041,E2 -3883.041} C_VEL
LIN {X 0,Y 539.378,Z 652.478,A -85,B 0,C 180,E1 -3883.324,E2 -3883.324} C_VEL
LIN {X 0,Y 539.524,Z 555.097,A -85,B 0,C 180,E1 -3884.639,E2 -3884.639} C_VEL
LIN {X 0,Y 538.369,Z 548.529,A -85,B 0,C 180,E1 -3884.77,E2 -3884.77} C_VEL
LIN {X 0,Y 538.267,Z 545.599,A -85,B 0,C 180,E1 -3885.137,E2 -3885.137} C_VEL
LIN {X 0,Y 538.441,Z 532.885,A -85,B 0,C 180,E1 -3887.469,E2 -3887.469} C_VEL
LIN {X 0,Y 538.624,Z 521.449,A -85,B 0,C 180,E1 -3889.632,E2 -3889.632} C_VEL
LIN {X 0,Y 538.064,Z 517.51,A -85,B 0,C 180,E1 -3890.458,E2 -3890.458} C_VEL
LIN {X 0,Y 538.024,Z 517.469,A -85,B 0,C 180,E1 -3893.071,E2 -3893.071} C_VEL
LIN {X 0,Y 538.044,Z 517.462,A -85,B 0,C 180,E1 -3895.672,E2 -3895.672} C_VEL
LIN {X 0,Y 538.046,Z 517.46,A -85,B 0,C 180,E1 -3898.049,E2 -3898.049} C_VEL
LIN {X 0,Y 538.02,Z 517.461,A -85,B 0,C 180,E1 -3900.626,E2 -3900.626} C_VEL
LIN {X 0,Y 538.044,Z 517.466,A -85,B 0,C 180,E1 -3903.282,E2 -3903.282} C_VEL
LIN {X 0,Y 538.026,Z 517.461,A -85,B 0,C 180,E1 -3906.001,E2 -3906.001} C_VEL
LIN {X 0,Y 538.014,Z 517.464,A -85,B 0,C 180,E1 -3908.829,E2 -3908.829} C_VEL
LIN {X 0,Y 538.035,Z 517.463,A -85,B 0,C 180,E1 -3911.879,E2 -3911.879} C_VEL
LIN {X 0,Y 538.028,Z 517.462,A -85,B 0,C 180,E1 -3915.14,E2 -3915.14} C_VEL
LIN {X 0,Y 538.037,Z 517.46,A -85,B 0,C 180,E1 -3918.227,E2 -3918.227} C_VEL
LIN {X 0,Y 538.055,Z 517.454,A -85,B 0,C 180,E1 -3920.411,E2 -3920.411} C_VEL
LIN {X 0,Y 538.028,Z 517.461,A -85,B 0,C 180,E1 -3923.067,E2 -3923.067} C_VEL
LIN {X 0,Y 538.028,Z 517.464,A -85,B 0,C 180,E1 -3925.827,E2 -3925.827} C_VEL
LIN {X 0,Y 538.019,Z 517.461,A -85,B 0,C 180,E1 -3928.499,E2 -3928.499} C_VEL
LIN {X 0,Y 538.053,Z 517.461,A -85,B 0,C 180,E1 -3931.099,E2 -3931.099} C_VEL
LIN {X 0,Y 538.045,Z 517.466,A -85,B 0,C 180,E1 -3933.633,E2 -3933.633} C_VEL
LIN {X 0,Y 538.016,Z 517.462,A -85,B 0,C 180,E1 -3936.118,E2 -3936.118} C_VEL
LIN {X 0,Y 538.036,Z 517.465,A -85,B 0,C 180,E1 -3939.348,E2 -3939.348} C_VEL
LIN {X 0,Y 538.066,Z 517.454,A -85,B 0,C 180,E1 -3942.517,E2 -3942.517} C_VEL
LIN {X 0,Y 538.057,Z 517.465,A -85,B 0,C 180,E1 -3945.63,E2 -3945.63} C_VEL
LIN {X 0,Y 538.07,Z 517.454,A -85,B 0,C 180,E1 -3948.701,E2 -3948.701} C_VEL
LIN {X 0,Y 538.083,Z 517.46,A -85,B 0,C 180,E1 -3951.739,E2 -3951.739} C_VEL
LIN {X 0,Y 538.158,Z 517.444,A -85,B 0,C 180,E1 -3954.755,E2 -3954.755} C_VEL
LIN {X 0,Y 538.161,Z 517.449,A -85,B 0,C 180,E1 -3957.755,E2 -3957.755} C_VEL
LIN {X 0,Y 538.178,Z 517.442,A -85,B 0,C 180,E1 -3960.748,E2 -3960.748} C_VEL
LIN {X 0,Y 538.136,Z 517.447,A -85,B 0,C 180,E1 -3962.994,E2 -3962.994} C_VEL
LIN {X 0,Y 538.117,Z 517.453,A -85,B 0,C 180,E1 -3965.997,E2 -3965.997} C_VEL
LIN {X 0,Y 538.065,Z 517.457,A -85,B 0,C 180,E1 -3969.018,E2 -3969.018} C_VEL
LIN {X 0,Y 538.076,Z 517.457,A -85,B 0,C 180,E1 -3972.063,E2 -3972.063} C_VEL
LIN {X 0,Y 538.038,Z 517.461,A -85,B 0,C 180,E1 -3975.144,E2 -3975.144} C_VEL
LIN {X 0,Y 538.028,Z 517.461,A -85,B 0,C 180,E1 -3978.27,E2 -3978.27} C_VEL
LIN {X 0,Y 538.036,Z 517.459,A -85,B 0,C 180,E1 -3980.652,E2 -3980.652} C_VEL
LIN {X 0,Y 538.017,Z 517.467,A -85,B 0,C 180,E1 -3983.888,E2 -3983.888} C_VEL
LIN {X 0,Y 538.044,Z 517.457,A -85,B 0,C 180,E1 -3986.367,E2 -3986.367} C_VEL
LIN {X 0,Y 538.026,Z 517.462,A -85,B 0,C 180,E1 -3988.934,E2 -3988.934} C_VEL
LIN {X 0,Y 538.022,Z 517.467,A -85,B 0,C 180,E1 -3991.891,E2 -3991.891} C_VEL
LIN {X 0,Y 538.029,Z 517.459,A -85,B 0,C 180,E1 -3994.622,E2 -3994.622} C_VEL
LIN {X 0,Y 538.002,Z 517.461,A -85,B 0,C 180,E1 -3997.171,E2 -3997.171} C_VEL
LIN {X 0,Y 538.025,Z 517.468,A -85,B 0,C 180,E1 -3999.797,E2 -3999.797} C_VEL
LIN {X 0,Y 538.015,Z 517.459,A -85,B 0,C 180,E1 -4002.787,E2 -4002.787} C_VEL
LIN {X 0,Y 538.026,Z 517.465,A -85,B 0,C 180,E1 -4005.926,E2 -4005.926} C_VEL
LIN {X 0,Y 538.075,Z 517.458,A -85,B 0,C 180,E1 -4009.25,E2 -4009.25} C_VEL
LIN {X 0,Y 537.992,Z 517.464,A -85,B 0,C 180,E1 -4012.123,E2 -4012.123} C_VEL
LIN {X 0,Y 538.01,Z 517.464,A -85,B 0,C 180,E1 -4014.918,E2 -4014.918} C_VEL
LIN {X 0,Y 538.03,Z 517.454,A -85,B 0,C 180,E1 -4017.619,E2 -4017.619} C_VEL
LIN {X 0,Y 538.017,Z 517.464,A -85,B 0,C 180,E1 -4020.24,E2 -4020.24} C_VEL
LIN {X 0,Y 538.065,Z 517.455,A -85,B 0,C 180,E1 -4022.797,E2 -4022.797} C_VEL
LIN {X 0,Y 538.031,Z 517.468,A -85,B 0,C 180,E1 -4025.704,E2 -4025.704} C_VEL
LIN {X 0,Y 538.101,Z 517.732,A -85,B 0,C 180,E1 -4026.158,E2 -4026.158} C_VEL
LIN {X 0,Y 539.343,Z 525.378,A -85,B 0,C 180,E1 -4027.435,E2 -4027.435} C_VEL
LIN {X 0,Y 538.924,Z 544.202,A -85,B 0,C 180,E1 -4030.38,E2 -4030.38} C_VEL
LIN {X 0,Y 538.56,Z 562.012,A -85,B 0,C 180,E1 -4033.122,E2 -4033.122} C_VEL
LIN {X 0,Y 538.39,Z 575.944,A -85,B 0,C 180,E1 -4035.222,E2 -4035.222} C_VEL
LIN {X 0,Y 539.233,Z 581.431,A -85,B 0,C 180,E1 -4035.348,E2 -4035.348} C_VEL
LIN {X 0,Y 539.698,Z 587.308,A -85,B 0,C 180,E1 -4035.44,E2 -4035.44} C_VEL
LIN {X 0,Y 539.349,Z 683.98,A -85,B 0,C 180,E1 -4036.748,E2 -4036.748} C_VEL
LIN {X 0,Y 539.149,Z 697.232,A -85,B 0,C 180,E1 -4037.078,E2 -4037.078} C_VEL
LIN {X 0,Y 538.951,Z 710.498,A -85,B 0,C 180,E1 -4037.576,E2 -4037.576} C_VEL
LIN {X 0,Y 538.744,Z 722.378,A -85,B 0,C 180,E1 -4038.189,E2 -4038.189} C_VEL
LIN {X 0,Y 538.515,Z 734.496,A -85,B 0,C 180,E1 -4038.997,E2 -4038.997} C_VEL
LIN {X 0,Y 538.228,Z 744.653,A -85,B 0,C 180,E1 -4039.848,E2 -4039.848} C_VEL
LIN {X 0,Y 538.026,Z 753.792,A -85,B 0,C 180,E1 -4040.793,E2 -4040.793} C_VEL
LIN {X 0,Y 537.85,Z 762.693,A -85,B 0,C 180,E1 -4041.926,E2 -4041.926} C_VEL
LIN {X 0,Y 537.728,Z 769.853,A -85,B 0,C 180,E1 -4043.057,E2 -4043.057} C_VEL
LIN {X 0,Y 537.676,Z 776.368,A -85,B 0,C 180,E1 -4044.375,E2 -4044.375} C_VEL
LIN {X 0,Y 537.557,Z 780.679,A -85,B 0,C 180,E1 -4045.502,E2 -4045.502} C_VEL
LIN {X 0,Y 537.591,Z 782.962,A -85,B 0,C 180,E1 -4046.253,E2 -4046.253} C_VEL
LIN {X 0,Y 537.551,Z 784.811,A -85,B 0,C 180,E1 -4047.003,E2 -4047.003} C_VEL
LIN {X 0,Y 537.451,Z 787.185,A -85,B 0,C 180,E1 -4048.502,E2 -4048.502} C_VEL
LIN {X 0,Y 537.442,Z 788,A -85,B 0,C 180,E1 -4050.001,E2 -4050.001} C_VEL
LIN {X 0,Y 537.451,Z 787.182,A -85,B 0,C 180,E1 -4051.499,E2 -4051.499} C_VEL
LIN {X 0,Y 537.551,Z 784.806,A -85,B 0,C 180,E1 -4052.998,E2 -4052.998} C_VEL
LIN {X 0,Y 537.603,Z 781.893,A -85,B 0,C 180,E1 -4054.124,E2 -4054.124} C_VEL
LIN {X 0,Y 537.588,Z 777.947,A -85,B 0,C 180,E1 -4055.251,E2 -4055.251} C_VEL
LIN {X 0,Y 537.65,Z 773.08,A -85,B 0,C 180,E1 -4056.335,E2 -4056.335} C_VEL
LIN {X 0,Y 537.791,Z 766.462,A -85,B 0,C 180,E1 -4057.51,E2 -4057.51} C_VEL
LIN {X 0,Y 537.973,Z 758.473,A -85,B 0,C 180,E1 -4058.641,E2 -4058.641} C_VEL
LIN {X 0,Y 538.144,Z 750.328,A -85,B 0,C 180,E1 -4059.586,E2 -4059.586} C_VEL
LIN {X 0,Y 538.34,Z 740.392,A -85,B 0,C 180,E1 -4060.532,E2 -4060.532} C_VEL
LIN {X 0,Y 538.577,Z 730.581,A -85,B 0,C 180,E1 -4061.288,E2 -4061.288} C_VEL
LIN {X 0,Y 538.754,Z 719.533,A -85,B 0,C 180,E1 -4061.974,E2 -4061.974} C_VEL
LIN {X 0,Y 539.002,Z 707.097,A -85,B 0,C 180,E1 -4062.568,E2 -4062.568} C_VEL
LIN {X 0,Y 539.222,Z 694.075,A -85,B 0,C 180,E1 -4063.017,E2 -4063.017} C_VEL
LIN {X 0,Y 539.377,Z 681.07,A -85,B 0,C 180,E1 -4063.301,E2 -4063.301} C_VEL
LIN {X 0,Y 539.57,Z 583.668,A -85,B 0,C 180,E1 -4064.612,E2 -4064.612} C_VEL
LIN {X 0,Y 538.384,Z 576.044,A -85,B 0,C 180,E1 -4064.771,E2 -4064.771} C_VEL
LIN {X 0,Y 538.693,Z 556.313,A -85,B 0,C 180,E1 -4067.751,E2 -4067.751} C_VEL
LIN {X 0,Y 539.09,Z 536.56,A -85,B 0,C 180,E1 -4070.809,E2 -4070.809} C_VEL
LIN {X 0,Y 539.263,Z 523.829,A -85,B 0,C 180,E1 -4072.813,E2 -4072.813} C_VEL
LIN {X 0,Y 538.038,Z 517.552,A -85,B 0,C 180,E1 -4073.913,E2 -4073.913} C_VEL
LIN {X 0,Y 538.046,Z 517.463,A -85,B 0,C 180,E1 -4076.367,E2 -4076.367} C_VEL
LIN {X 0,Y 538.034,Z 517.456,A -85,B 0,C 180,E1 -4078.934,E2 -4078.934} C_VEL
LIN {X 0,Y 538.014,Z 517.468,A -85,B 0,C 180,E1 -4081.887,E2 -4081.887} C_VEL
LIN {X 0,Y 538.016,Z 517.466,A -85,B 0,C 180,E1 -4084.618,E2 -4084.618} C_VEL
LIN {X 0,Y 538.008,Z 517.464,A -85,B 0,C 180,E1 -4087.17,E2 -4087.17} C_VEL
LIN {X 0,Y 538.026,Z 517.465,A -85,B 0,C 180,E1 -4089.797,E2 -4089.797} C_VEL
LIN {X 0,Y 538.023,Z 517.464,A -85,B 0,C 180,E1 -4092.786,E2 -4092.786} C_VEL
LIN {X 0,Y 538.011,Z 517.464,A -85,B 0,C 180,E1 -4095.138,E2 -4095.138} C_VEL
LIN {X 0,Y 538.033,Z 517.469,A -85,B 0,C 180,E1 -4098.227,E2 -4098.227} C_VEL
LIN {X 0,Y 538.017,Z 517.463,A -85,B 0,C 180,E1 -4101.17,E2 -4101.17} C_VEL
LIN {X 0,Y 538.027,Z 517.469,A -85,B 0,C 180,E1 -4104.084,E2 -4104.084} C_VEL
LIN {X 0,Y 538.034,Z 517.464,A -85,B 0,C 180,E1 -4106.727,E2 -4106.727} C_VEL
LIN {X 0,Y 538.03,Z 517.464,A -85,B 0,C 180,E1 -4109.556,E2 -4109.556} C_VEL
LIN {X 0,Y 538.049,Z 517.466,A -85,B 0,C 180,E1 -4111.951,E2 -4111.951} C_VEL
LIN {X 0,Y 538.094,Z 517.59,A -85,B 0,C 180,E1 -4114.753,E2 -4114.753} C_VEL
LIN {X 0,Y 539.439,Z 525.606,A -85,B 0,C 180,E1 -4115.895,E2 -4115.895} C_VEL
LIN {X 0,Y 539.197,Z 545.763,A -85,B 0,C 180,E1 -4118.595,E2 -4118.595} C_VEL
LIN {X 0,Y 538.907,Z 565.779,A -85,B 0,C 180,E1 -4121.367,E2 -4121.367} C_VEL
LIN {X 0,Y 538.583,Z 584.002,A -85,B 0,C 180,E1 -4123.901,E2 -4123.901} C_VEL
LIN {X 0,Y 538.305,Z 603.236,A -85,B 0,C 180,E1 -4126.6,E2 -4126.6} C_VEL
LIN {X 0,Y 538.119,Z 616.426,A -85,B 0,C 180,E1 -4128.411,E2 -4128.411} C_VEL
LIN {X 0,Y 538.834,Z 624.533,A -85,B 0,C 180,E1 -4128.557,E2 -4128.557} C_VEL
LIN {X 0,Y 538.703,Z 695.845,A -85,B 0,C 180,E1 -4129.524,E2 -4129.524} C_VEL
LIN {X 0,Y 538.568,Z 706.818,A -85,B 0,C 180,E1 -4129.806,E2 -4129.806} C_VEL
LIN {X 0,Y 538.417,Z 717.64,A -85,B 0,C 180,E1 -4130.23,E2 -4130.23} C_VEL
LIN {X 0,Y 538.254,Z 728.097,A -85,B 0,C 180,E1 -4130.796,E2 -4130.796} C_VEL
LIN {X 0,Y 538.109,Z 737.48,A -85,B 0,C 180,E1 -4131.456,E2 -4131.456} C_VEL
LIN {X 0,Y 537.927,Z 746.884,A -85,B 0,C 180,E1 -4132.304,E2 -4132.304} C_VEL
LIN {X 0,Y 537.825,Z 755.318,A -85,B 0,C 180,E1 -4133.279,E2 -4133.279} C_VEL
LIN {X 0,Y 537.768,Z 761.551,A -85,B 0,C 180,E1 -4134.187,E2 -4134.187} C_VEL
LIN {X 0,Y 537.605,Z 766.73,A -85,B 0,C 180,E1 -4135.126,E2 -4135.126} C_VEL
LIN {X 0,Y 537.6,Z 771.463,A -85,B 0,C 180,E1 -4136.252,E2 -4136.252} C_VEL
LIN {X 0,Y 537.564,Z 773.823,A -85,B 0,C 180,E1 -4137.002,E2 -4137.002} C_VEL
LIN {X 0,Y 537.489,Z 775.62,A -85,B 0,C 180,E1 -4137.752,E2 -4137.752} C_VEL
LIN {X 0,Y 537.449,Z 776.913,A -85,B 0,C 180,E1 -4138.501,E2 -4138.501} C_VEL
LIN {X 0,Y 537.439,Z 777.707,A -85,B 0,C 180,E1 -4139.251,E2 -4139.251} C_VEL
LIN {X 0,Y 537.44,Z 777.996,A -85,B 0,C 180,E1 -4140,E2 -4140} C_VEL
LIN {X 0,Y 537.44,Z 777.776,A -85,B 0,C 180,E1 -4140.749,E2 -4140.749} C_VEL
LIN {X 0,Y 537.452,Z 777.043,A -85,B 0,C 180,E1 -4141.499,E2 -4141.499} C_VEL
LIN {X 0,Y 537.491,Z 775.803,A -85,B 0,C 180,E1 -4142.248,E2 -4142.248} C_VEL
LIN {X 0,Y 537.59,Z 772.986,A -85,B 0,C 180,E1 -4143.373,E2 -4143.373} C_VEL
LIN {X 0,Y 537.606,Z 768.864,A -85,B 0,C 180,E1 -4144.499,E2 -4144.499} C_VEL
LIN {X 0,Y 537.71,Z 763.234,A -85,B 0,C 180,E1 -4145.626,E2 -4145.626} C_VEL
LIN {X 0,Y 537.786,Z 756.29,A -85,B 0,C 180,E1 -4146.685,E2 -4146.685} C_VEL
LIN {X 0,Y 537.884,Z 749.529,A -85,B 0,C 180,E1 -4147.508,E2 -4147.508} C_VEL
LIN {X 0,Y 538.039,Z 740.858,A -85,B 0,C 180,E1 -4148.356,E2 -4148.356} C_VEL
LIN {X 0,Y 538.293,Z 730.985,A -85,B 0,C 180,E1 -4149.109,E2 -4149.109} C_VEL
LIN {X 0,Y 538.401,Z 721.421,A -85,B 0,C 180,E1 -4149.675,E2 -4149.675} C_VEL
LIN {X 0,Y 538.569,Z 710.786,A -85,B 0,C 180,E1 -4150.147,E2 -4150.147} C_VEL
LIN {X 0,Y 538.633,Z 699.035,A -85,B 0,C 180,E1 -4150.502,E2 -4150.502} C_VEL
LIN {X 0,Y 538.745,Z 684.494,A -85,B 0,C 180,E1 -4150.737,E2 -4150.737} C_VEL
LIN {X 0,Y 538.714,Z 621.65,A -85,B 0,C 180,E1 -4151.574,E2 -4151.574} C_VEL
